RoboDK station: kr30 cnc template amana 46348 - paulina work pls TOO LOW AAA 2.rdk

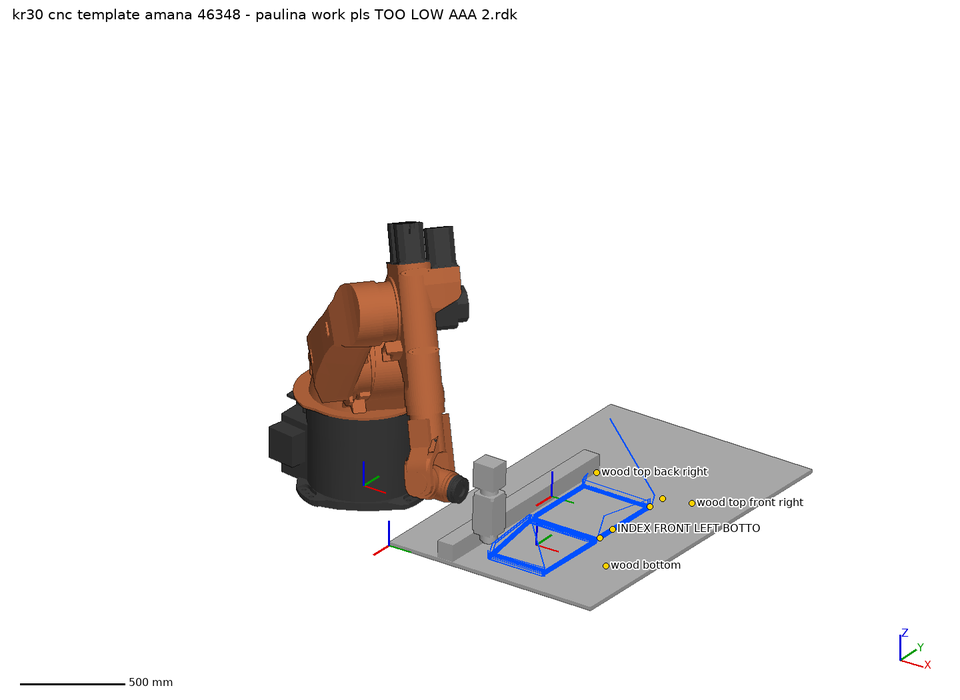
[picture v0: the station drawn from its stored meshes, robots at their saved joint values, targets as dots, program paths as lines]
Station kr30 cnc template amana 46348 - paulina work pls TOO LOW AAA 2. Poses are relative to the parent item; angles as X-Y-Z fixed-axis rotations.
  - frame KUKA KR 30 HA Base at (0, 0, 0) mm
    - robot KUKA KR 30 HA: 6 axes, payload 30 kg, reach 2033 mm, repeatability 0.05 mm, weight 665 kg
        modified DH rows (alpha deg, a mm, theta deg, d mm): 0, 0, 0, 815; -90, 350, 0, 0; 0, 850, -90, 0; -90, 145, 0, 820; 90, 0, 0, 0; -90, 0, 180, 170
        joint limits [-185, -135, -120, -350, -119, -350] to [185, 35, 158, 350, 119, 350]; home [0, -90, 90, 0, 0, 0]; saved at [41.891, -43.185, 108.764, -135.148, 71.183, 163.257]
      - tool rc90 spindle mm, TCP at (267.95, 0.68, 160.99) mm, rotated rx 0 ry 90 rz 0 deg, size 110 x 421.3 x 118 mm, geometry from rc90 spindle mm.stl
    - frame Tabletop at (921.82, -1104.91, 385) mm, rotated rx -0.93 ry -0.21 rz -89.9 deg
      - object tabletop CHECK HEIGHT at (-1839.9, 0, 0) mm, size 1839.9 x 1168.4 x 19 mm, geometry from kr30 tabletop mm.stl
      - object kr30 pipe jig base at (-1220, -610.6, 0) mm, size 1217.6 x 88.9 x 88.9 mm, geometry from kr30 pipe jig base.stl
      - frame Frame 3 at (-820, 370, 45) mm
        - frame Frame 4 at (470, 240, 0) mm, rotated rx 0 ry 0 rz 90 deg
      - target wood top back right (Cartesian target) at (-1141.49, 406.84, 52.26) mm, rotated rx 18.07 ry 89.88 rz 108.17 deg; joints [-2.086, -55.392, 143.759, 178.106, 87.553, -179.775] of KUKA KR 30 HA
      - target wood bottom (Cartesian target) at (-376.62, 995.52, 35.89) mm, rotated rx 18.07 ry 89.88 rz 108.17 deg; joints [24.587, -27.296, 76.752, 211.623, 53.064, -199.759] of KUKA KR 30 HA
      - target wood top front right (Cartesian target) at (-1142.68, 960.22, 52.55) mm, rotated rx 18.06 ry 89.88 rz 108.16 deg; joints [-1.42, -37.516, 98.016, 178.579, 59.693, -179.129] of KUKA KR 30 HA
      - target INDEX FRONT LEFT BOTTOM OF CUT (Cartesian target) at (-711.64, 800.54, 39.36) mm, rotated rx 179.19 ry 0.89 rz -118.74 deg; joints [9.3, -40.938, 107.706, -20.874, -68.324, 7.9] of KUKA KR 30 HA
      - target index front right bottom (Cartesian target) at (-1126.88, 801.86, 37.54) mm, rotated rx -179.93 ry 1.1 rz -61.86 deg; joints [5.389, -41.179, 108.718, 35.697, -71.625, -13.066] of KUKA KR 30 HA
    - target new front left bottom (Cartesian target) at (1722.92, -500.67, 408.01) mm, rotated rx 179.79 ry 0.28 rz -161.47 deg; joints [23.344, -37.525, 99.802, 45.258, -69.995, -19.505] of KUKA KR 30 HA
    - target new front right bottom (Cartesian target) at (1723.89, -86.44, 408.76) mm, rotated rx 179.79 ry 0.28 rz -161.47 deg; joints [7.822, -41.869, 110.032, 28.03, -70.804, -10.277] of KUKA KR 30 HA
  - machining project Machining Settings: C:/Users/Research Office/Desktop/paulina a5.apt | rotZ(0) | rotX(0)*rotY(0) | rotZ(0)
  - machining project Machining Settings2: C:/Users/Research Office/Desktop/paulina wooorrkkk.apt | rotZ(0) | rotX(0)*rotY(0) | rotz(0) | onStart | onPathStart | onApproach | onPoint | onRetract | onFinish | onPathFinish
  - program Machining (2349 instructions, listed below)
  - program Machining (769 instructions, listed below)
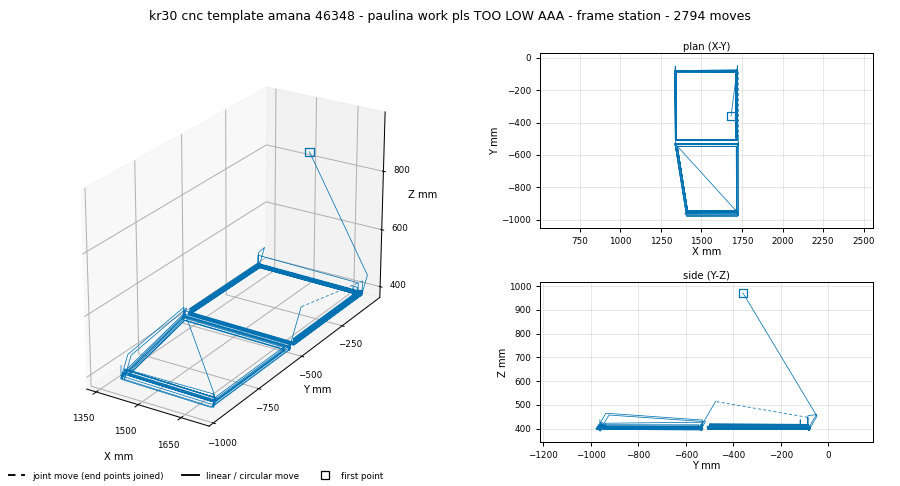
[picture p0: tool path of kr30 cnc template amana 46348 - paulina work pls TOO LOW AAA 2.rdk in frame station, 2794 of 2794 moves have a stored position in this frame; points joined in program order, loops and branches not executed]

--- program Machining (robot KUKA KR 30 HA) ---
  Smooth(15)
  Print: /'1001'
  Print: /''
  Print: /'diagonal cut'
  Set speed (100.0 mm/s)
  Set Ref.: Frame 3
  Set Tool: rc90 spindle mm
  Show rc90 spindle mm
  MoveJ 1 to (78.48, 382.25, 556.62) mm, rotated rx 174.11 ry -15.54 rz -70.77 deg; joints [17.697, -62.551, 89.928, 80.197, -35.892, -71.862]
  MoveL 2 to (-235.36, 431, 39.15) mm, rotated rx -174.06 ry -29.54 rz -11.91 deg; joints [6.63, -38.675, 85.378, -71.398, 65.68, 136.343]
  MoveL 3 to (-235.36, 431, 39.15) mm, rotated rx -174.06 ry -29.54 rz -11.91 deg; joints [6.63, -38.675, 85.378, -71.398, 65.68, 136.343]
  Set speed (100.0 mm/s)
  MoveL 4 to (-206.65, 431, -10.41) mm, rotated rx -174.06 ry -29.54 rz -11.91 deg; joints [7.609, -36.412, 85.1, -71.619, 65.676, 138.638]
  Set speed (38.1 mm/s)
  MoveL 5 to (-201.55, 431, -19.21) mm, rotated rx -174.06 ry -29.54 rz -11.91 deg; joints [7.783, -35.998, 85.023, -71.649, 65.678, 139.029]
  MoveL 6 to (-200.68, 431, -19.44) mm, rotated rx -174.06 ry -29.54 rz -11.91 deg; joints [7.812, -35.981, 85.01, -71.631, 65.695, 139.038]
  Set speed (76.2 mm/s)
  MoveL 7 to (-202.44, 431, -12.48) mm, rotated rx -174.06 ry -29.54 rz -11.91 deg; joints [7.751, -36.293, 85.037, -71.549, 65.747, 138.728]
  MoveL 8 to (-201.13, 431, -12.23) mm, rotated rx -174.06 ry -29.54 rz -11.91 deg; joints [7.795, -36.294, 85.017, -71.511, 65.781, 138.716]
  MoveL 9 to (-196.56, 431, -16.91) mm, rotated rx -174.06 ry -29.54 rz -11.91 deg; joints [7.95, -36.06, 84.947, -71.479, 65.826, 138.922]
  Set speed (38.1 mm/s)
  MoveL 10 to (-196.33, 431, -16.04) mm, rotated rx -174.06 ry -29.54 rz -11.91 deg; joints [7.958, -36.095, 84.943, -71.457, 65.843, 138.883]
  Set speed (100.0 mm/s)
  MoveL 11 to (-203.65, 431, -3.41) mm, rotated rx -174.06 ry -29.54 rz -11.91 deg; joints [7.709, -36.688, 85.05, -71.414, 65.842, 138.321]
  MoveL 12 to (-199.05, 427.82, -0.75) mm, rotated rx -174.06 ry -29.54 rz -11.91 deg; joints [7.878, -36.942, 85.328, -71.314, 65.94, 138.386]
  Set speed (38.1 mm/s)
  MoveL 13 to (-197.47, 427.82, -3.47) mm, rotated rx -174.06 ry -29.54 rz -11.91 deg; joints [7.932, -36.814, 85.306, -71.324, 65.94, 138.508]
  MoveL 14 to (-197.39, 427.82, -3.84) mm, rotated rx -174.06 ry -29.54 rz -11.91 deg; joints [7.935, -36.798, 85.305, -71.328, 65.937, 138.525]
  Set speed (76.2 mm/s)
  MoveL 15 to (-197.71, 427.82, -8.22) mm, rotated rx -174.06 ry -29.54 rz -11.91 deg; joints [7.925, -36.614, 85.314, -71.416, 65.869, 138.722]
  MoveL 16 to (-199.91, 427.82, -8.42) mm, rotated rx -174.06 ry -29.54 rz -11.91 deg; joints [7.851, -36.621, 85.348, -71.477, 65.815, 138.733]
  MoveL 17 to (-206.05, 427.82, -11.57) mm, rotated rx -174.06 ry -29.54 rz -11.91 deg; joints [7.644, -36.531, 85.443, -71.692, 65.627, 138.878]
  MoveL 18 to (-201.08, 427.82, -20.25) mm, rotated rx -174.06 ry -29.54 rz -11.91 deg; joints [7.814, -36.122, 85.367, -71.723, 65.628, 139.265]
  MoveL 19 to (-201.08, 424.65, -20.25) mm, rotated rx -174.06 ry -29.54 rz -11.91 deg; joints [7.829, -36.293, 85.717, -71.79, 65.581, 139.454]
  MoveL 20 to (-206.05, 424.65, -11.57) mm, rotated rx -174.06 ry -29.54 rz -11.91 deg; joints [7.659, -36.704, 85.792, -71.758, 65.581, 139.066]
  MoveL 21 to (-200.05, 424.65, -8.41) mm, rotated rx -174.06 ry -29.54 rz -11.91 deg; joints [7.861, -36.796, 85.7, -71.545, 65.765, 138.92]
  MoveL 22 to (-197.85, 424.65, -8.4) mm, rotated rx -174.06 ry -29.54 rz -11.91 deg; joints [7.935, -36.78, 85.666, -71.488, 65.817, 138.918]
  MoveL 23 to (-197.85, 424.65, -4.14) mm, rotated rx -174.06 ry -29.54 rz -11.91 deg; joints [7.935, -36.962, 85.662, -71.41, 65.875, 138.725]
  Set speed (38.1 mm/s)
  MoveL 24 to (-197.89, 424.65, -3.98) mm, rotated rx -174.06 ry -29.54 rz -11.91 deg; joints [7.933, -36.969, 85.663, -71.408, 65.877, 138.718]
  MoveL 25 to (-198.05, 424.33, -3.7) mm, rotated rx -174.06 ry -29.54 rz -11.91 deg; joints [7.929, -36.999, 85.7, -71.414, 65.872, 138.724]
  Set speed (76.2 mm/s)
  MoveL 26 to (-198.05, 421.79, -3.7) mm, rotated rx -174.06 ry -29.54 rz -11.91 deg; joints [7.941, -37.137, 85.979, -71.466, 65.835, 138.873]
  Set speed (38.1 mm/s)
  MoveL 27 to (-197.89, 421.47, -3.98) mm, rotated rx -174.06 ry -29.54 rz -11.91 deg; joints [7.948, -37.142, 86.011, -71.473, 65.83, 138.904]
  MoveL 28 to (-197.85, 421.47, -4.14) mm, rotated rx -174.06 ry -29.54 rz -11.91 deg; joints [7.95, -37.135, 86.011, -71.475, 65.829, 138.911]
  Set speed (76.2 mm/s)
  MoveL 29 to (-197.85, 421.47, -8.28) mm, rotated rx -174.06 ry -29.54 rz -11.91 deg; joints [7.951, -36.957, 86.014, -71.551, 65.772, 139.099]
  MoveL 30 to (-200, 421.47, -8.41) mm, rotated rx -174.06 ry -29.54 rz -11.91 deg; joints [7.878, -36.968, 86.047, -71.61, 65.72, 139.107]
  MoveL 31 to (-206.05, 421.47, -11.57) mm, rotated rx -174.06 ry -29.54 rz -11.91 deg; joints [7.673, -36.876, 86.14, -71.825, 65.535, 139.254]
  MoveL 32 to (-201.08, 421.47, -20.25) mm, rotated rx -174.06 ry -29.54 rz -11.91 deg; joints [7.844, -36.464, 86.065, -71.856, 65.535, 139.642]
  MoveL 33 to (-201.08, 418.3, -20.25) mm, rotated rx -174.06 ry -29.54 rz -11.91 deg; joints [7.859, -36.635, 86.412, -71.923, 65.489, 139.83]
  MoveL 34 to (-206.05, 418.3, -11.57) mm, rotated rx -174.06 ry -29.54 rz -11.91 deg; joints [7.688, -37.047, 86.487, -71.891, 65.489, 139.44]
  MoveL 35 to (-199.95, 418.3, -8.41) mm, rotated rx -174.06 ry -29.54 rz -11.91 deg; joints [7.895, -37.139, 86.394, -71.673, 65.675, 139.293]
  MoveL 36 to (-197.85, 418.3, -8.16) mm, rotated rx -174.06 ry -29.54 rz -11.91 deg; joints [7.966, -37.134, 86.361, -71.614, 65.728, 139.28]
  MoveL 37 to (-197.85, 418.3, -4.14) mm, rotated rx -174.06 ry -29.54 rz -11.91 deg; joints [7.965, -37.307, 86.358, -71.54, 65.783, 139.097]
  Set speed (38.1 mm/s)
  MoveL 38 to (-197.89, 418.3, -3.98) mm, rotated rx -174.06 ry -29.54 rz -11.91 deg; joints [7.963, -37.314, 86.359, -71.538, 65.784, 139.09]
  MoveL 39 to (-198.05, 417.98, -3.7) mm, rotated rx -174.06 ry -29.54 rz -11.91 deg; joints [7.96, -37.344, 86.395, -71.543, 65.779, 139.096]
  Set speed (76.2 mm/s)
  MoveL 40 to (-198.05, 415.44, -3.7) mm, rotated rx -174.06 ry -29.54 rz -11.91 deg; joints [7.972, -37.481, 86.672, -71.595, 65.743, 139.244]
  Set speed (38.1 mm/s)
  MoveL 41 to (-197.89, 415.12, -3.98) mm, rotated rx -174.06 ry -29.54 rz -11.91 deg; joints [7.979, -37.485, 86.704, -71.602, 65.738, 139.275]
  MoveL 42 to (-197.85, 415.12, -4.14) mm, rotated rx -174.06 ry -29.54 rz -11.91 deg; joints [7.98, -37.478, 86.704, -71.604, 65.737, 139.282]
  Set speed (76.2 mm/s)
  MoveL 43 to (-197.85, 415.12, -8.4) mm, rotated rx -174.06 ry -29.54 rz -11.91 deg; joints [7.981, -37.294, 86.707, -71.683, 65.679, 139.477]
  MoveL 44 to (-199.9, 415.12, -8.41) mm, rotated rx -174.06 ry -29.54 rz -11.91 deg; joints [7.911, -37.309, 86.739, -71.737, 65.631, 139.478]
  MoveL 45 to (-206.05, 415.12, -11.57) mm, rotated rx -174.06 ry -29.54 rz -11.91 deg; joints [7.703, -37.217, 86.833, -71.957, 65.444, 139.627]
  MoveL 46 to (-201.08, 415.12, -20.25) mm, rotated rx -174.06 ry -29.54 rz -11.91 deg; joints [7.874, -36.804, 86.758, -71.989, 65.444, 140.017]
  MoveL 47 to (-201.08, 411.95, -20.25) mm, rotated rx -174.06 ry -29.54 rz -11.91 deg; joints [7.889, -36.973, 87.102, -72.055, 65.399, 140.204]
  MoveL 48 to (-206.05, 411.95, -11.57) mm, rotated rx -174.06 ry -29.54 rz -11.91 deg; joints [7.718, -37.387, 87.177, -72.023, 65.399, 139.812]
  MoveL 49 to (-199.84, 411.95, -8.41) mm, rotated rx -174.06 ry -29.54 rz -11.91 deg; joints [7.928, -37.479, 87.082, -71.801, 65.587, 139.663]
  MoveL 50 to (-197.85, 411.95, -8.4) mm, rotated rx -174.06 ry -29.54 rz -11.91 deg; joints [7.996, -37.465, 87.052, -71.748, 65.634, 139.662]
  MoveL 51 to (-197.85, 411.95, -4.14) mm, rotated rx -174.06 ry -29.54 rz -11.91 deg; joints [7.996, -37.649, 87.048, -71.668, 65.692, 139.466]
  Set speed (38.1 mm/s)
  MoveL 52 to (-197.89, 411.95, -3.98) mm, rotated rx -174.06 ry -29.54 rz -11.91 deg; joints [7.994, -37.656, 87.049, -71.666, 65.693, 139.459]
  MoveL 53 to (-198.05, 411.63, -3.7) mm, rotated rx -174.06 ry -29.54 rz -11.91 deg; joints [7.99, -37.686, 87.085, -71.672, 65.689, 139.465]
  Set speed (76.2 mm/s)
  MoveL 54 to (-198.05, 409.09, -3.7) mm, rotated rx -174.06 ry -29.54 rz -11.91 deg; joints [8.002, -37.822, 87.36, -71.723, 65.653, 139.612]
  Set speed (38.1 mm/s)
  MoveL 55 to (-197.89, 408.77, -3.98) mm, rotated rx -174.06 ry -29.54 rz -11.91 deg; joints [8.009, -37.826, 87.392, -71.73, 65.648, 139.643]
  MoveL 56 to (-197.85, 408.77, -4.14) mm, rotated rx -174.06 ry -29.54 rz -11.91 deg; joints [8.011, -37.819, 87.391, -71.732, 65.647, 139.65]
  Set speed (76.2 mm/s)
  MoveL 57 to (-197.85, 408.77, -8.4) mm, rotated rx -174.06 ry -29.54 rz -11.91 deg; joints [8.012, -37.634, 87.395, -71.813, 65.589, 139.846]
  MoveL 58 to (-200.19, 408.77, -8.41) mm, rotated rx -174.06 ry -29.54 rz -11.91 deg; joints [7.932, -37.651, 87.431, -71.874, 65.534, 139.848]
  MoveL 59 to (-206.05, 408.77, -11.57) mm, rotated rx -174.06 ry -29.54 rz -11.91 deg; joints [7.733, -37.556, 87.52, -72.089, 65.355, 139.997]
  MoveL 60 to (-201.08, 408.77, -20.25) mm, rotated rx -174.06 ry -29.54 rz -11.91 deg; joints [7.904, -37.141, 87.445, -72.121, 65.355, 140.39]
  MoveL 61 to (-201.08, 405.6, -20.25) mm, rotated rx -174.06 ry -29.54 rz -11.91 deg; joints [7.919, -37.309, 87.787, -72.187, 65.311, 140.576]
  MoveL 62 to (-206.05, 405.6, -11.57) mm, rotated rx -174.06 ry -29.54 rz -11.91 deg; joints [7.747, -37.724, 87.862, -72.154, 65.31, 140.182]
  MoveL 63 to (-200.12, 405.6, -8.41) mm, rotated rx -174.06 ry -29.54 rz -11.91 deg; joints [7.949, -37.819, 87.771, -71.937, 65.491, 140.032]
  MoveL 64 to (-197.85, 405.6, -8.4) mm, rotated rx -174.06 ry -29.54 rz -11.91 deg; joints [8.027, -37.803, 87.737, -71.877, 65.544, 140.03]
  MoveL 65 to (-197.85, 405.6, -4.14) mm, rotated rx -174.06 ry -29.54 rz -11.91 deg; joints [8.026, -37.988, 87.733, -71.796, 65.602, 139.833]
  MoveL 66 to (-197.85, 405.47, -3.66) mm, rotated rx -174.06 ry -29.54 rz -11.91 deg; joints [8.027, -38.015, 87.747, -71.79, 65.607, 139.819]
  MoveL 67 to (-197.85, 405.12, -3.31) mm, rotated rx -174.06 ry -29.54 rz -11.91 deg; joints [8.029, -38.049, 87.784, -71.79, 65.607, 139.823]
  MoveL 68 to (-197.85, 404.64, -3.19) mm, rotated rx -174.06 ry -29.54 rz -11.91 deg; joints [8.031, -38.08, 87.835, -71.797, 65.602, 139.844]
  MoveL 69 to (-197.85, 403.37, -3.19) mm, rotated rx -174.06 ry -29.54 rz -11.91 deg; joints [8.037, -38.147, 87.971, -71.823, 65.585, 139.917]
  MoveL 70 to (-197.85, 402.9, -3.31) mm, rotated rx -174.06 ry -29.54 rz -11.91 deg; joints [8.039, -38.167, 88.022, -71.835, 65.576, 139.951]
  MoveL 71 to (-197.85, 402.55, -3.66) mm, rotated rx -174.06 ry -29.54 rz -11.91 deg; joints [8.041, -38.171, 88.06, -71.848, 65.567, 139.987]
  MoveL 72 to (-197.85, 402.42, -4.14) mm, rotated rx -174.06 ry -29.54 rz -11.91 deg; joints [8.042, -38.157, 88.074, -71.86, 65.558, 140.016]
  MoveL 73 to (-197.85, 402.42, -8.4) mm, rotated rx -174.06 ry -29.54 rz -11.91 deg; joints [8.043, -37.972, 88.077, -71.941, 65.5, 140.213]
  MoveL 74 to (-200.05, 402.42, -8.41) mm, rotated rx -174.06 ry -29.54 rz -11.91 deg; joints [7.967, -37.987, 88.111, -72, 65.449, 140.215]
  MoveL 75 to (-206.05, 402.42, -11.57) mm, rotated rx -174.06 ry -29.54 rz -11.91 deg; joints [7.762, -37.892, 88.202, -72.22, 65.267, 140.366]
  MoveL 76 to (-201.08, 402.42, -20.25) mm, rotated rx -174.06 ry -29.54 rz -11.91 deg; joints [7.935, -37.476, 88.128, -72.252, 65.267, 140.761]
  MoveL 77 to (-201.08, 399.25, -20.25) mm, rotated rx -174.06 ry -29.54 rz -11.91 deg; joints [7.95, -37.642, 88.467, -72.318, 65.223, 140.946]
  MoveL 78 to (-206.05, 399.25, -11.57) mm, rotated rx -174.06 ry -29.54 rz -11.91 deg; joints [7.777, -38.059, 88.541, -72.285, 65.224, 140.55]
  MoveL 79 to (-199.98, 399.25, -8.41) mm, rotated rx -174.06 ry -29.54 rz -11.91 deg; joints [7.985, -38.154, 88.449, -72.062, 65.407, 140.398]
  MoveL 80 to (-197.85, 399.25, -8.4) mm, rotated rx -174.06 ry -29.54 rz -11.91 deg; joints [8.058, -38.139, 88.416, -72.005, 65.457, 140.396]
  MoveL 81 to (-197.85, 399.25, -4.14) mm, rotated rx -174.06 ry -29.54 rz -11.91 deg; joints [8.057, -38.325, 88.413, -71.923, 65.515, 140.198]
  Set speed (38.1 mm/s)
  MoveL 82 to (-197.89, 399.25, -3.98) mm, rotated rx -174.06 ry -29.54 rz -11.91 deg; joints [8.056, -38.332, 88.414, -71.922, 65.516, 140.191]
  MoveL 83 to (-198.05, 398.93, -3.7) mm, rotated rx -174.06 ry -29.54 rz -11.91 deg; joints [8.052, -38.362, 88.45, -71.927, 65.511, 140.197]
  Set speed (76.2 mm/s)
  MoveL 84 to (-198.05, 396.39, -3.7) mm, rotated rx -174.06 ry -29.54 rz -11.91 deg; joints [8.064, -38.496, 88.72, -71.978, 65.477, 140.342]
  Set speed (38.1 mm/s)
  MoveL 85 to (-197.89, 396.07, -3.98) mm, rotated rx -174.06 ry -29.54 rz -11.91 deg; joints [8.072, -38.5, 88.752, -71.985, 65.472, 140.373]
  MoveL 86 to (-197.85, 396.07, -4.14) mm, rotated rx -174.06 ry -29.54 rz -11.91 deg; joints [8.073, -38.492, 88.751, -71.987, 65.471, 140.38]
  Set speed (76.2 mm/s)
  MoveL 87 to (-197.85, 396.07, -8.4) mm, rotated rx -174.06 ry -29.54 rz -11.91 deg; joints [8.074, -38.306, 88.755, -72.068, 65.413, 140.578]
  MoveL 88 to (-199.91, 396.07, -8.41) mm, rotated rx -174.06 ry -29.54 rz -11.91 deg; joints [8.003, -38.321, 88.786, -72.124, 65.365, 140.581]
  MoveL 89 to (-206.05, 396.07, -11.57) mm, rotated rx -174.06 ry -29.54 rz -11.91 deg; joints [7.793, -38.226, 88.879, -72.35, 65.181, 140.733]
  MoveL 90 to (-201.08, 396.07, -20.25) mm, rotated rx -174.06 ry -29.54 rz -11.91 deg; joints [7.965, -37.808, 88.805, -72.383, 65.181, 141.13]
  MoveL 91 to (-201.08, 392.9, -20.25) mm, rotated rx -174.06 ry -29.54 rz -11.91 deg; joints [7.981, -37.973, 89.142, -72.448, 65.138, 141.314]
  MoveL 92 to (-206.05, 392.9, -11.57) mm, rotated rx -174.06 ry -29.54 rz -11.91 deg; joints [7.808, -38.392, 89.216, -72.415, 65.138, 140.915]
  MoveL 93 to (-199.84, 392.9, -8.41) mm, rotated rx -174.06 ry -29.54 rz -11.91 deg; joints [8.021, -38.487, 89.122, -72.186, 65.324, 140.762]
  MoveL 94 to (-197.85, 392.9, -8.38) mm, rotated rx -174.06 ry -29.54 rz -11.91 deg; joints [8.09, -38.473, 89.091, -72.132, 65.371, 140.759]
  MoveL 95 to (-197.85, 392.9, -4.14) mm, rotated rx -174.06 ry -29.54 rz -11.91 deg; joints [8.089, -38.659, 89.088, -72.05, 65.428, 140.561]
  Set speed (38.1 mm/s)
  MoveL 96 to (-197.89, 392.9, -3.98) mm, rotated rx -174.06 ry -29.54 rz -11.91 deg; joints [8.087, -38.666, 89.089, -72.048, 65.43, 140.554]
  MoveL 97 to (-198.05, 392.58, -3.7) mm, rotated rx -174.06 ry -29.54 rz -11.91 deg; joints [8.083, -38.696, 89.124, -72.053, 65.425, 140.559]
  Set speed (76.2 mm/s)
  MoveL 98 to (-198.05, 390.04, -3.7) mm, rotated rx -174.06 ry -29.54 rz -11.91 deg; joints [8.096, -38.829, 89.393, -72.104, 65.391, 140.704]
  Set speed (38.1 mm/s)
  MoveL 99 to (-197.89, 389.72, -3.98) mm, rotated rx -174.06 ry -29.54 rz -11.91 deg; joints [8.103, -38.833, 89.424, -72.111, 65.387, 140.734]
  MoveL 100 to (-197.85, 389.72, -4.14) mm, rotated rx -174.06 ry -29.54 rz -11.91 deg; joints [8.104, -38.825, 89.424, -72.113, 65.386, 140.742]
  Set speed (76.2 mm/s)
  MoveL 101 to (-197.85, 389.72, -8.26) mm, rotated rx -174.06 ry -29.54 rz -11.91 deg; joints [8.105, -38.645, 89.427, -72.193, 65.33, 140.935]
  MoveL 102 to (-199.77, 389.72, -8.41) mm, rotated rx -174.06 ry -29.54 rz -11.91 deg; joints [8.039, -38.652, 89.456, -72.248, 65.283, 140.944]
  MoveL 103 to (-206.05, 389.72, -11.57) mm, rotated rx -174.06 ry -29.54 rz -11.91 deg; joints [7.823, -38.557, 89.551, -72.48, 65.096, 141.097]
  MoveL 104 to (-201.08, 389.72, -20.25) mm, rotated rx -174.06 ry -29.54 rz -11.91 deg; joints [7.996, -38.138, 89.477, -72.513, 65.096, 141.497]
  MoveL 105 to (-201.08, 386.55, -20.25) mm, rotated rx -174.06 ry -29.54 rz -11.91 deg; joints [8.012, -38.302, 89.811, -72.578, 65.054, 141.679]
  MoveL 106 to (-206.05, 386.55, -11.57) mm, rotated rx -174.06 ry -29.54 rz -11.91 deg; joints [7.838, -38.722, 89.885, -72.545, 65.054, 141.278]
  MoveL 107 to (-199.7, 386.55, -8.41) mm, rotated rx -174.06 ry -29.54 rz -11.91 deg; joints [8.057, -38.817, 89.79, -72.31, 65.243, 141.124]
  MoveL 108 to (-197.85, 386.55, -8.41) mm, rotated rx -174.06 ry -29.54 rz -11.91 deg; joints [8.121, -38.803, 89.762, -72.259, 65.286, 141.122]
  MoveL 109 to (-197.85, 386.55, -4.14) mm, rotated rx -174.06 ry -29.54 rz -11.91 deg; joints [8.12, -38.991, 89.758, -72.176, 65.344, 140.922]
  Set speed (38.1 mm/s)
  MoveL 110 to (-197.89, 386.55, -3.98) mm, rotated rx -174.06 ry -29.54 rz -11.91 deg; joints [8.119, -38.998, 89.759, -72.174, 65.345, 140.914]
  MoveL 111 to (-198.05, 386.23, -3.7) mm, rotated rx -174.06 ry -29.54 rz -11.91 deg; joints [8.115, -39.028, 89.794, -72.179, 65.341, 140.92]
  Set speed (76.2 mm/s)
  MoveL 112 to (-198.05, 383.69, -3.7) mm, rotated rx -174.06 ry -29.54 rz -11.91 deg; joints [8.127, -39.16, 90.061, -72.229, 65.307, 141.063]
  Set speed (38.1 mm/s)
  MoveL 113 to (-197.89, 383.37, -3.98) mm, rotated rx -174.06 ry -29.54 rz -11.91 deg; joints [8.135, -39.163, 90.092, -72.237, 65.303, 141.094]
  MoveL 114 to (-197.85, 383.37, -4.14) mm, rotated rx -174.06 ry -29.54 rz -11.91 deg; joints [8.136, -39.156, 90.092, -72.239, 65.302, 141.102]
  Set speed (76.2 mm/s)
  MoveL 115 to (-197.85, 383.37, -8.4) mm, rotated rx -174.06 ry -29.54 rz -11.91 deg; joints [8.137, -38.968, 90.095, -72.322, 65.244, 141.302]
  MoveL 116 to (-199.66, 383.37, -8.41) mm, rotated rx -174.06 ry -29.54 rz -11.91 deg; joints [8.074, -38.981, 90.122, -72.372, 65.202, 141.305]
  MoveL 117 to (-206.05, 383.37, -11.57) mm, rotated rx -174.06 ry -29.54 rz -11.91 deg; joints [7.854, -38.886, 90.218, -72.609, 65.013, 141.459]
  MoveL 118 to (-201.08, 383.37, -20.25) mm, rotated rx -174.06 ry -29.54 rz -11.91 deg; joints [8.028, -38.465, 90.145, -72.642, 65.012, 141.861]
  MoveL 119 to (-201.08, 380.2, -20.25) mm, rotated rx -174.06 ry -29.54 rz -11.91 deg; joints [8.043, -38.628, 90.477, -72.707, 64.971, 142.043]
  MoveL 120 to (-206.05, 380.2, -11.57) mm, rotated rx -174.06 ry -29.54 rz -11.91 deg; joints [7.869, -39.05, 90.55, -72.673, 64.972, 141.64]
  MoveL 121 to (-200.12, 380.2, -8.41) mm, rotated rx -174.06 ry -29.54 rz -11.91 deg; joints [8.074, -39.148, 90.461, -72.447, 65.15, 141.485]
  MoveL 122 to (-197.85, 380.2, -8.4) mm, rotated rx -174.06 ry -29.54 rz -11.91 deg; joints [8.153, -39.132, 90.427, -72.385, 65.203, 141.482]
  MoveL 123 to (-197.85, 380.2, -4.14) mm, rotated rx -174.06 ry -29.54 rz -11.91 deg; joints [8.152, -39.321, 90.424, -72.301, 65.26, 141.281]
  Set speed (38.1 mm/s)
  MoveL 124 to (-197.89, 380.2, -3.98) mm, rotated rx -174.06 ry -29.54 rz -11.91 deg; joints [8.151, -39.328, 90.424, -72.299, 65.261, 141.273]
  MoveL 125 to (-198.05, 379.88, -3.7) mm, rotated rx -174.06 ry -29.54 rz -11.91 deg; joints [8.147, -39.358, 90.459, -72.304, 65.257, 141.278]
  Set speed (76.2 mm/s)
  MoveL 126 to (-198.05, 377.34, -3.7) mm, rotated rx -174.06 ry -29.54 rz -11.91 deg; joints [8.159, -39.489, 90.724, -72.354, 65.224, 141.421]
  Set speed (38.1 mm/s)
  MoveL 127 to (-197.89, 377.02, -3.98) mm, rotated rx -174.06 ry -29.54 rz -11.91 deg; joints [8.166, -39.492, 90.755, -72.361, 65.22, 141.452]
  MoveL 128 to (-197.85, 377.02, -4.14) mm, rotated rx -174.06 ry -29.54 rz -11.91 deg; joints [8.168, -39.485, 90.755, -72.363, 65.219, 141.459]
  Set speed (76.2 mm/s)
  MoveL 129 to (-197.85, 377.02, -8.4) mm, rotated rx -174.06 ry -29.54 rz -11.91 deg; joints [8.169, -39.296, 90.758, -72.448, 65.161, 141.661]
  MoveL 130 to (-200.07, 377.02, -8.41) mm, rotated rx -174.06 ry -29.54 rz -11.91 deg; joints [8.092, -39.311, 90.791, -72.509, 65.11, 141.664]
  MoveL 131 to (-206.05, 377.02, -11.57) mm, rotated rx -174.06 ry -29.54 rz -11.91 deg; joints [7.884, -39.213, 90.881, -72.737, 64.931, 141.82]
  MoveL 132 to (-201.08, 377.02, -20.25) mm, rotated rx -174.06 ry -29.54 rz -11.91 deg; joints [8.059, -38.79, 90.808, -72.771, 64.93, 142.224]
  MoveL 133 to (-201.08, 373.85, -20.25) mm, rotated rx -174.06 ry -29.54 rz -11.91 deg; joints [8.075, -38.951, 91.137, -72.835, 64.89, 142.404]
  MoveL 134 to (-206.05, 373.85, -11.57) mm, rotated rx -174.06 ry -29.54 rz -11.91 deg; joints [7.9, -39.375, 91.211, -72.801, 64.891, 141.999]
  MoveL 135 to (-200.58, 373.85, -8.41) mm, rotated rx -174.06 ry -29.54 rz -11.91 deg; joints [8.09, -39.478, 91.129, -72.586, 65.058, 141.843]
  MoveL 136 to (-197.85, 373.85, -8.4) mm, rotated rx -174.06 ry -29.54 rz -11.91 deg; joints [8.185, -39.459, 91.088, -72.51, 65.121, 141.84]
  MoveL 137 to (-197.85, 373.85, -4.14) mm, rotated rx -174.06 ry -29.54 rz -11.91 deg; joints [8.184, -39.648, 91.084, -72.426, 65.178, 141.637]
  Set speed (38.1 mm/s)
  MoveL 138 to (-197.89, 373.85, -3.98) mm, rotated rx -174.06 ry -29.54 rz -11.91 deg; joints [8.183, -39.655, 91.085, -72.424, 65.179, 141.63]
  MoveL 139 to (-198.05, 373.53, -3.7) mm, rotated rx -174.06 ry -29.54 rz -11.91 deg; joints [8.179, -39.685, 91.12, -72.429, 65.175, 141.635]
  Set speed (76.2 mm/s)
  MoveL 140 to (-198.05, 370.99, -3.7) mm, rotated rx -174.06 ry -29.54 rz -11.91 deg; joints [8.191, -39.815, 91.383, -72.478, 65.143, 141.777]
  Set speed (38.1 mm/s)
  MoveL 141 to (-197.89, 370.67, -3.98) mm, rotated rx -174.06 ry -29.54 rz -11.91 deg; joints [8.199, -39.818, 91.414, -72.486, 65.139, 141.807]
  MoveL 142 to (-197.85, 370.67, -4.14) mm, rotated rx -174.06 ry -29.54 rz -11.91 deg; joints [8.2, -39.811, 91.413, -72.488, 65.138, 141.815]
  Set speed (76.2 mm/s)
  MoveL 143 to (-197.85, 370.67, -8.4) mm, rotated rx -174.06 ry -29.54 rz -11.91 deg; joints [8.201, -39.621, 91.416, -72.572, 65.08, 142.018]
  MoveL 144 to (-200.55, 370.67, -8.41) mm, rotated rx -174.06 ry -29.54 rz -11.91 deg; joints [8.107, -39.64, 91.457, -72.648, 65.018, 142.022]
  MoveL 145 to (-206.05, 370.67, -11.57) mm, rotated rx -174.06 ry -29.54 rz -11.91 deg; joints [7.915, -39.537, 91.539, -72.865, 64.851, 142.178]
  MoveL 146 to (-201.08, 370.67, -20.25) mm, rotated rx -174.06 ry -29.54 rz -11.91 deg; joints [8.091, -39.112, 91.466, -72.899, 64.85, 142.584]
  MoveL 147 to (-201.08, 367.5, -20.25) mm, rotated rx -174.06 ry -29.54 rz -11.91 deg; joints [8.107, -39.273, 91.794, -72.963, 64.81, 142.764]
  MoveL 148 to (-206.05, 367.5, -11.57) mm, rotated rx -174.06 ry -29.54 rz -11.91 deg; joints [7.931, -39.699, 91.867, -72.929, 64.811, 142.357]
  MoveL 149 to (-200.51, 367.5, -8.41) mm, rotated rx -174.06 ry -29.54 rz -11.91 deg; joints [8.124, -39.801, 91.784, -72.71, 64.979, 142.2]
  MoveL 150 to (-197.85, 367.5, -8.4) mm, rotated rx -174.06 ry -29.54 rz -11.91 deg; joints [8.217, -39.783, 91.744, -72.635, 65.04, 142.196]
  MoveL 151 to (-197.85, 367.5, -4.14) mm, rotated rx -174.06 ry -29.54 rz -11.91 deg; joints [8.216, -39.973, 91.741, -72.549, 65.098, 141.992]
  MoveL 152 to (-197.85, 367.37, -3.66) mm, rotated rx -174.06 ry -29.54 rz -11.91 deg; joints [8.217, -40.001, 91.753, -72.542, 65.103, 141.976]
  MoveL 153 to (-197.85, 367.02, -3.31) mm, rotated rx -174.06 ry -29.54 rz -11.91 deg; joints [8.219, -40.034, 91.789, -72.542, 65.103, 141.979]
  MoveL 154 to (-197.85, 366.55, -3.19) mm, rotated rx -174.06 ry -29.54 rz -11.91 deg; joints [8.221, -40.064, 91.838, -72.549, 65.099, 142]
  MoveL 155 to (-197.85, 365.28, -3.19) mm, rotated rx -174.06 ry -29.54 rz -11.91 deg; joints [8.227, -40.129, 91.968, -72.574, 65.083, 142.07]
  MoveL 156 to (-197.85, 364.8, -3.31) mm, rotated rx -174.06 ry -29.54 rz -11.91 deg; joints [8.23, -40.147, 92.018, -72.585, 65.075, 142.103]
  MoveL 157 to (-197.85, 364.45, -3.66) mm, rotated rx -174.06 ry -29.54 rz -11.91 deg; joints [8.232, -40.15, 92.054, -72.599, 65.066, 142.139]
  MoveL 158 to (-197.85, 364.33, -4.14) mm, rotated rx -174.06 ry -29.54 rz -11.91 deg; joints [8.233, -40.135, 92.067, -72.611, 65.058, 142.169]
  MoveL 159 to (-197.85, 364.33, -8.4) mm, rotated rx -174.06 ry -29.54 rz -11.91 deg; joints [8.233, -39.944, 92.07, -72.697, 65.001, 142.373]
  MoveL 160 to (-200.48, 364.33, -8.41) mm, rotated rx -174.06 ry -29.54 rz -11.91 deg; joints [8.141, -39.962, 92.11, -72.771, 64.94, 142.377]
  MoveL 161 to (-206.05, 364.33, -11.57) mm, rotated rx -174.06 ry -29.54 rz -11.91 deg; joints [7.947, -39.859, 92.193, -72.992, 64.772, 142.535]
  MoveL 162 to (-201.08, 364.33, -20.25) mm, rotated rx -174.06 ry -29.54 rz -11.91 deg; joints [8.123, -39.433, 92.12, -73.026, 64.771, 142.943]
  MoveL 163 to (-201.08, 361.15, -20.25) mm, rotated rx -174.06 ry -29.54 rz -11.91 deg; joints [8.139, -39.592, 92.445, -73.09, 64.732, 143.122]
  MoveL 164 to (-206.05, 361.15, -11.57) mm, rotated rx -174.06 ry -29.54 rz -11.91 deg; joints [7.962, -40.02, 92.518, -73.055, 64.733, 142.712]
  MoveL 165 to (-200.44, 361.15, -8.41) mm, rotated rx -174.06 ry -29.54 rz -11.91 deg; joints [8.159, -40.123, 92.435, -72.832, 64.902, 142.554]
  MoveL 166 to (-197.85, 361.15, -8.4) mm, rotated rx -174.06 ry -29.54 rz -11.91 deg; joints [8.25, -40.105, 92.396, -72.759, 64.961, 142.55]
  MoveL 167 to (-197.85, 361.15, -4.14) mm, rotated rx -174.06 ry -29.54 rz -11.91 deg; joints [8.249, -40.296, 92.393, -72.673, 65.018, 142.345]
  Set speed (38.1 mm/s)
  MoveL 168 to (-197.89, 361.15, -3.98) mm, rotated rx -174.06 ry -29.54 rz -11.91 deg; joints [8.247, -40.303, 92.393, -72.671, 65.02, 142.337]
  MoveL 169 to (-198.05, 360.83, -3.7) mm, rotated rx -174.06 ry -29.54 rz -11.91 deg; joints [8.243, -40.333, 92.428, -72.676, 65.016, 142.342]
  Set speed (76.2 mm/s)
  MoveL 170 to (-198.05, 358.29, -3.7) mm, rotated rx -174.06 ry -29.54 rz -11.91 deg; joints [8.256, -40.462, 92.687, -72.725, 64.984, 142.483]
  Set speed (38.1 mm/s)
  MoveL 171 to (-197.89, 357.98, -3.98) mm, rotated rx -174.06 ry -29.54 rz -11.91 deg; joints [8.264, -40.464, 92.718, -72.732, 64.981, 142.513]
  MoveL 172 to (-197.85, 357.98, -4.14) mm, rotated rx -174.06 ry -29.54 rz -11.91 deg; joints [8.265, -40.457, 92.717, -72.734, 64.979, 142.521]
  Set speed (76.2 mm/s)
  MoveL 173 to (-197.85, 357.98, -8.25) mm, rotated rx -174.06 ry -29.54 rz -11.91 deg; joints [8.266, -40.272, 92.72, -72.817, 64.924, 142.719]
  MoveL 174 to (-200.41, 357.98, -8.41) mm, rotated rx -174.06 ry -29.54 rz -11.91 deg; joints [8.176, -40.283, 92.759, -72.893, 64.864, 142.73]
  MoveL 175 to (-206.05, 357.98, -11.57) mm, rotated rx -174.06 ry -29.54 rz -11.91 deg; joints [7.978, -40.179, 92.843, -73.118, 64.694, 142.889]
  MoveL 176 to (-201.08, 357.98, -20.25) mm, rotated rx -174.06 ry -29.54 rz -11.91 deg; joints [8.155, -39.751, 92.77, -73.153, 64.693, 143.3]
  MoveL 177 to (-201.08, 354.8, -20.25) mm, rotated rx -174.06 ry -29.54 rz -11.91 deg; joints [8.171, -39.909, 93.093, -73.216, 64.655, 143.478]
  MoveL 178 to (-206.05, 354.8, -11.57) mm, rotated rx -174.06 ry -29.54 rz -11.91 deg; joints [7.994, -40.339, 93.166, -73.181, 64.656, 143.066]
  MoveL 179 to (-200.37, 354.8, -8.41) mm, rotated rx -174.06 ry -29.54 rz -11.91 deg; joints [8.193, -40.442, 93.081, -72.954, 64.826, 142.906]
  MoveL 180 to (-197.85, 354.8, -8.13) mm, rotated rx -174.06 ry -29.54 rz -11.91 deg; joints [8.282, -40.437, 93.043, -72.877, 64.887, 142.889]
  MoveL 181 to (-197.85, 354.8, -4.14) mm, rotated rx -174.06 ry -29.54 rz -11.91 deg; joints [8.282, -40.617, 93.04, -72.795, 64.941, 142.696]
  MoveL 182 to (-197.85, 354.67, -3.66) mm, rotated rx -174.06 ry -29.54 rz -11.91 deg; joints [8.282, -40.645, 93.053, -72.788, 64.945, 142.68]
  MoveL 183 to (-197.85, 354.32, -3.31) mm, rotated rx -174.06 ry -29.54 rz -11.91 deg; joints [8.284, -40.678, 93.088, -72.788, 64.946, 142.682]
  MoveL 184 to (-197.85, 353.85, -3.19) mm, rotated rx -174.06 ry -29.54 rz -11.91 deg; joints [8.286, -40.708, 93.136, -72.794, 64.942, 142.702]
  MoveL 185 to (-197.85, 352.58, -3.19) mm, rotated rx -174.06 ry -29.54 rz -11.91 deg; joints [8.293, -40.771, 93.265, -72.819, 64.926, 142.772]
  MoveL 186 to (-197.85, 352.1, -3.31) mm, rotated rx -174.06 ry -29.54 rz -11.91 deg; joints [8.295, -40.79, 93.314, -72.83, 64.919, 142.805]
  MoveL 187 to (-197.85, 351.75, -3.66) mm, rotated rx -174.06 ry -29.54 rz -11.91 deg; joints [8.297, -40.791, 93.349, -72.844, 64.91, 142.841]
  MoveL 188 to (-197.85, 351.63, -4.14) mm, rotated rx -174.06 ry -29.54 rz -11.91 deg; joints [8.298, -40.776, 93.363, -72.856, 64.902, 142.871]
  MoveL 189 to (-197.85, 351.63, -8.4) mm, rotated rx -174.06 ry -29.54 rz -11.91 deg; joints [8.299, -40.584, 93.366, -72.944, 64.845, 143.078]
  MoveL 190 to (-200.34, 351.63, -8.41) mm, rotated rx -174.06 ry -29.54 rz -11.91 deg; joints [8.211, -40.601, 93.403, -73.015, 64.788, 143.082]
  MoveL 191 to (-206.05, 351.63, -11.57) mm, rotated rx -174.06 ry -29.54 rz -11.91 deg; joints [8.01, -40.497, 93.488, -73.244, 64.618, 143.242]
  MoveL 192 to (-201.08, 351.63, -20.25) mm, rotated rx -174.06 ry -29.54 rz -11.91 deg; joints [8.187, -40.067, 93.415, -73.279, 64.616, 143.656]
  MoveL 193 to (-201.08, 348.45, -20.25) mm, rotated rx -174.06 ry -29.54 rz -11.91 deg; joints [8.204, -40.224, 93.736, -73.342, 64.579, 143.833]
  MoveL 194 to (-206.05, 348.45, -11.57) mm, rotated rx -174.06 ry -29.54 rz -11.91 deg; joints [8.026, -40.655, 93.809, -73.307, 64.58, 143.418]
  MoveL 195 to (-199.95, 348.45, -8.41) mm, rotated rx -174.06 ry -29.54 rz -11.91 deg; joints [8.241, -40.757, 93.718, -73.066, 64.759, 143.256]
  MoveL 196 to (-197.85, 348.45, -8.4) mm, rotated rx -174.06 ry -29.54 rz -11.91 deg; joints [8.316, -40.742, 93.687, -73.005, 64.807, 143.253]
  MoveL 197 to (-197.85, 348.45, -4.14) mm, rotated rx -174.06 ry -29.54 rz -11.91 deg; joints [8.315, -40.935, 93.684, -72.917, 64.864, 143.045]
  MoveL 198 to (-197.85, 348.32, -3.66) mm, rotated rx -174.06 ry -29.54 rz -11.91 deg; joints [8.315, -40.963, 93.696, -72.91, 64.869, 143.029]
  MoveL 199 to (-197.85, 347.98, -3.31) mm, rotated rx -174.06 ry -29.54 rz -11.91 deg; joints [8.317, -40.997, 93.731, -72.909, 64.869, 143.031]
  MoveL 200 to (-197.85, 347.5, -3.19) mm, rotated rx -174.06 ry -29.54 rz -11.91 deg; joints [8.319, -41.026, 93.779, -72.916, 64.865, 143.051]
  MoveL 201 to (-197.85, 346.23, -3.19) mm, rotated rx -174.06 ry -29.54 rz -11.91 deg; joints [8.326, -41.09, 93.907, -72.94, 64.85, 143.121]
  MoveL 202 to (-197.85, 345.75, -3.31) mm, rotated rx -174.06 ry -29.54 rz -11.91 deg; joints [8.329, -41.108, 93.955, -72.952, 64.843, 143.153]
  MoveL 203 to (-197.85, 345.4, -3.66) mm, rotated rx -174.06 ry -29.54 rz -11.91 deg; joints [8.33, -41.109, 93.991, -72.966, 64.834, 143.189]
  MoveL 204 to (-197.85, 345.28, -4.14) mm, rotated rx -174.06 ry -29.54 rz -11.91 deg; joints [8.331, -41.094, 94.004, -72.978, 64.826, 143.219]
  MoveL 205 to (-197.85, 345.28, -8.4) mm, rotated rx -174.06 ry -29.54 rz -11.91 deg; joints [8.332, -40.9, 94.007, -73.066, 64.769, 143.428]
  MoveL 206 to (-199.91, 345.28, -8.41) mm, rotated rx -174.06 ry -29.54 rz -11.91 deg; joints [8.259, -40.915, 94.038, -73.126, 64.722, 143.431]
  MoveL 207 to (-206.05, 345.28, -11.57) mm, rotated rx -174.06 ry -29.54 rz -11.91 deg; joints [8.042, -40.813, 94.129, -73.369, 64.543, 143.594]
  MoveL 208 to (-201.08, 345.28, -20.25) mm, rotated rx -174.06 ry -29.54 rz -11.91 deg; joints [8.22, -40.381, 94.056, -73.405, 64.541, 144.009]
  MoveL 209 to (-201.08, 342.1, -20.25) mm, rotated rx -174.06 ry -29.54 rz -11.91 deg; joints [8.237, -40.537, 94.376, -73.467, 64.504, 144.185]
  MoveL 210 to (-206.05, 342.1, -11.57) mm, rotated rx -174.06 ry -29.54 rz -11.91 deg; joints [8.058, -40.97, 94.448, -73.431, 64.506, 143.769]
  MoveL 211 to (-199.87, 342.1, -8.41) mm, rotated rx -174.06 ry -29.54 rz -11.91 deg; joints [8.277, -41.072, 94.357, -73.186, 64.686, 143.605]
  MoveL 212 to (-197.85, 342.1, -8.4) mm, rotated rx -174.06 ry -29.54 rz -11.91 deg; joints [8.349, -41.058, 94.327, -73.127, 64.732, 143.602]
  MoveL 213 to (-197.85, 342.1, -4.14) mm, rotated rx -174.06 ry -29.54 rz -11.91 deg; joints [8.348, -41.252, 94.323, -73.038, 64.789, 143.393]
  Set speed (38.1 mm/s)
  MoveL 214 to (-197.89, 342.1, -3.98) mm, rotated rx -174.06 ry -29.54 rz -11.91 deg; joints [8.346, -41.26, 94.324, -73.036, 64.79, 143.385]
  MoveL 215 to (-198.05, 341.78, -3.7) mm, rotated rx -174.06 ry -29.54 rz -11.91 deg; joints [8.342, -41.289, 94.358, -73.041, 64.786, 143.389]
  Set speed (76.2 mm/s)
  MoveL 216 to (-198.05, 339.25, -3.7) mm, rotated rx -174.06 ry -29.54 rz -11.91 deg; joints [8.356, -41.415, 94.612, -73.09, 64.757, 143.528]
  Set speed (38.1 mm/s)
  MoveL 217 to (-197.89, 338.93, -3.98) mm, rotated rx -174.06 ry -29.54 rz -11.91 deg; joints [8.363, -41.417, 94.642, -73.097, 64.753, 143.558]
  MoveL 218 to (-197.85, 338.93, -4.14) mm, rotated rx -174.06 ry -29.54 rz -11.91 deg; joints [8.365, -41.41, 94.642, -73.099, 64.752, 143.566]
  Set speed (76.2 mm/s)
  MoveL 219 to (-197.85, 338.93, -8.4) mm, rotated rx -174.06 ry -29.54 rz -11.91 deg; joints [8.366, -41.215, 94.645, -73.188, 64.695, 143.776]
  MoveL 220 to (-200.2, 338.93, -8.41) mm, rotated rx -174.06 ry -29.54 rz -11.91 deg; joints [8.282, -41.231, 94.68, -73.257, 64.642, 143.779]
  MoveL 221 to (-206.05, 338.93, -11.57) mm, rotated rx -174.06 ry -29.54 rz -11.91 deg; joints [8.074, -41.127, 94.766, -73.494, 64.469, 143.943]
  MoveL 222 to (-201.08, 338.93, -20.25) mm, rotated rx -174.06 ry -29.54 rz -11.91 deg; joints [8.253, -40.693, 94.694, -73.529, 64.467, 144.361]
  MoveL 223 to (-201.08, 335.75, -20.25) mm, rotated rx -174.06 ry -29.54 rz -11.91 deg; joints [8.27, -40.848, 95.011, -73.592, 64.431, 144.536]
  MoveL 224 to (-206.05, 335.75, -11.57) mm, rotated rx -174.06 ry -29.54 rz -11.91 deg; joints [8.091, -41.283, 95.083, -73.556, 64.432, 144.117]
  MoveL 225 to (-200.15, 335.75, -8.41) mm, rotated rx -174.06 ry -29.54 rz -11.91 deg; joints [8.3, -41.388, 94.996, -73.316, 64.606, 143.953]
  MoveL 226 to (-197.85, 335.75, -8.4) mm, rotated rx -174.06 ry -29.54 rz -11.91 deg; joints [8.382, -41.372, 94.962, -73.248, 64.658, 143.949]
  MoveL 227 to (-197.85, 335.75, -4.14) mm, rotated rx -174.06 ry -29.54 rz -11.91 deg; joints [8.381, -41.567, 94.959, -73.159, 64.715, 143.739]
  Set speed (38.1 mm/s)
  MoveL 228 to (-197.89, 335.75, -3.98) mm, rotated rx -174.06 ry -29.54 rz -11.91 deg; joints [8.38, -41.574, 94.959, -73.157, 64.716, 143.731]
  MoveL 229 to (-198.05, 335.44, -3.7) mm, rotated rx -174.06 ry -29.54 rz -11.91 deg; joints [8.376, -41.604, 94.993, -73.162, 64.712, 143.735]
  Set speed (76.2 mm/s)
  MoveL 230 to (-198.05, 332.9, -3.7) mm, rotated rx -174.06 ry -29.54 rz -11.91 deg; joints [8.389, -41.729, 95.246, -73.21, 64.683, 143.873]
  Set speed (38.1 mm/s)
  MoveL 231 to (-197.89, 332.58, -3.98) mm, rotated rx -174.06 ry -29.54 rz -11.91 deg; joints [8.397, -41.731, 95.276, -73.217, 64.679, 143.903]
  MoveL 232 to (-197.85, 332.58, -4.14) mm, rotated rx -174.06 ry -29.54 rz -11.91 deg; joints [8.398, -41.723, 95.275, -73.219, 64.678, 143.911]
  Set speed (76.2 mm/s)
  MoveL 233 to (-197.85, 332.58, -8.4) mm, rotated rx -174.06 ry -29.54 rz -11.91 deg; joints [8.399, -41.528, 95.278, -73.309, 64.621, 144.122]
  MoveL 234 to (-200.15, 332.58, -8.41) mm, rotated rx -174.06 ry -29.54 rz -11.91 deg; joints [8.317, -41.544, 95.312, -73.377, 64.57, 144.126]
  MoveL 235 to (-206.05, 332.58, -11.57) mm, rotated rx -174.06 ry -29.54 rz -11.91 deg; joints [8.107, -41.439, 95.399, -73.617, 64.396, 144.291]
  MoveL 236 to (-201.08, 332.58, -20.25) mm, rotated rx -174.06 ry -29.54 rz -11.91 deg; joints [8.286, -41.003, 95.327, -73.654, 64.395, 144.711]
  MoveL 237 to (-201.08, 329.4, -20.25) mm, rotated rx -174.06 ry -29.54 rz -11.91 deg; joints [8.303, -41.157, 95.642, -73.715, 64.359, 144.885]
  MoveL 238 to (-206.05, 329.4, -11.57) mm, rotated rx -174.06 ry -29.54 rz -11.91 deg; joints [8.123, -41.594, 95.715, -73.679, 64.36, 144.464]
  MoveL 239 to (-200.15, 329.4, -8.41) mm, rotated rx -174.06 ry -29.54 rz -11.91 deg; joints [8.334, -41.699, 95.628, -73.437, 64.533, 144.298]
  MoveL 240 to (-197.85, 329.4, -8.4) mm, rotated rx -174.06 ry -29.54 rz -11.91 deg; joints [8.416, -41.683, 95.594, -73.369, 64.585, 144.295]
  MoveL 241 to (-197.85, 329.4, -4.14) mm, rotated rx -174.06 ry -29.54 rz -11.91 deg; joints [8.415, -41.88, 95.59, -73.279, 64.642, 144.083]
  Set speed (38.1 mm/s)
  MoveL 242 to (-197.89, 329.4, -3.98) mm, rotated rx -174.06 ry -29.54 rz -11.91 deg; joints [8.414, -41.887, 95.591, -73.277, 64.643, 144.075]
  MoveL 243 to (-198.05, 329.09, -3.7) mm, rotated rx -174.06 ry -29.54 rz -11.91 deg; joints [8.41, -41.917, 95.624, -73.282, 64.64, 144.079]
  Set speed (76.2 mm/s)
  MoveL 244 to (-198.05, 326.55, -3.7) mm, rotated rx -174.06 ry -29.54 rz -11.91 deg; joints [8.423, -42.041, 95.876, -73.33, 64.611, 144.216]
  Set speed (38.1 mm/s)
  MoveL 245 to (-197.89, 326.23, -3.98) mm, rotated rx -174.06 ry -29.54 rz -11.91 deg; joints [8.431, -42.043, 95.905, -73.337, 64.607, 144.246]
  MoveL 246 to (-197.85, 326.23, -4.14) mm, rotated rx -174.06 ry -29.54 rz -11.91 deg; joints [8.432, -42.035, 95.905, -73.339, 64.606, 144.254]
  Set speed (76.2 mm/s)
  MoveL 247 to (-197.85, 326.23, -8.4) mm, rotated rx -174.06 ry -29.54 rz -11.91 deg; joints [8.433, -41.839, 95.908, -73.429, 64.549, 144.467]
  MoveL 248 to (-200.15, 326.23, -8.41) mm, rotated rx -174.06 ry -29.54 rz -11.91 deg; joints [8.351, -41.854, 95.942, -73.498, 64.498, 144.471]
  MoveL 249 to (-206.05, 326.23, -11.57) mm, rotated rx -174.06 ry -29.54 rz -11.91 deg; joints [8.14, -41.749, 96.029, -73.741, 64.325, 144.637]
  MoveL 250 to (-201.08, 326.23, -20.25) mm, rotated rx -174.06 ry -29.54 rz -11.91 deg; joints [8.32, -41.31, 95.957, -73.777, 64.323, 145.059]
  MoveL 251 to (-201.08, 323.05, -20.25) mm, rotated rx -174.06 ry -29.54 rz -11.91 deg; joints [8.337, -41.464, 96.27, -73.839, 64.288, 145.233]
  MoveL 252 to (-206.05, 323.05, -11.57) mm, rotated rx -174.06 ry -29.54 rz -11.91 deg; joints [8.156, -41.903, 96.342, -73.802, 64.29, 144.809]
  MoveL 253 to (-200.15, 323.05, -8.41) mm, rotated rx -174.06 ry -29.54 rz -11.91 deg; joints [8.367, -42.009, 96.255, -73.558, 64.462, 144.642]
  MoveL 254 to (-197.85, 323.05, -8.4) mm, rotated rx -174.06 ry -29.54 rz -11.91 deg; joints [8.45, -41.993, 96.221, -73.489, 64.514, 144.638]
  MoveL 255 to (-197.85, 323.05, -4.14) mm, rotated rx -174.06 ry -29.54 rz -11.91 deg; joints [8.449, -42.19, 96.218, -73.398, 64.57, 144.425]
  Set speed (38.1 mm/s)
  MoveL 256 to (-197.89, 323.05, -3.98) mm, rotated rx -174.06 ry -29.54 rz -11.91 deg; joints [8.448, -42.198, 96.219, -73.396, 64.571, 144.417]
  MoveL 257 to (-198.05, 322.74, -3.7) mm, rotated rx -174.06 ry -29.54 rz -11.91 deg; joints [8.444, -42.227, 96.252, -73.401, 64.568, 144.421]
  Set speed (76.2 mm/s)
  MoveL 258 to (-198.05, 320.2, -3.7) mm, rotated rx -174.06 ry -29.54 rz -11.91 deg; joints [8.457, -42.351, 96.502, -73.449, 64.54, 144.557]
  Set speed (38.1 mm/s)
  MoveL 259 to (-197.89, 319.88, -3.98) mm, rotated rx -174.06 ry -29.54 rz -11.91 deg; joints [8.465, -42.353, 96.531, -73.456, 64.536, 144.588]
  MoveL 260 to (-197.85, 319.88, -4.14) mm, rotated rx -174.06 ry -29.54 rz -11.91 deg; joints [8.467, -42.345, 96.531, -73.458, 64.535, 144.596]
  Set speed (76.2 mm/s)
  MoveL 261 to (-197.85, 319.88, -8.4) mm, rotated rx -174.06 ry -29.54 rz -11.91 deg; joints [8.467, -42.147, 96.534, -73.549, 64.478, 144.81]
  MoveL 262 to (-200.15, 319.88, -8.41) mm, rotated rx -174.06 ry -29.54 rz -11.91 deg; joints [8.384, -42.163, 96.568, -73.618, 64.427, 144.814]
  MoveL 263 to (-206.05, 319.88, -11.57) mm, rotated rx -174.06 ry -29.54 rz -11.91 deg; joints [8.173, -42.057, 96.655, -73.863, 64.255, 144.981]
  MoveL 264 to (-201.08, 319.88, -20.25) mm, rotated rx -174.06 ry -29.54 rz -11.91 deg; joints [8.354, -41.617, 96.583, -73.9, 64.253, 145.406]
  MoveL 265 to (-201.08, 316.7, -20.25) mm, rotated rx -174.06 ry -29.54 rz -11.91 deg; joints [8.371, -41.769, 96.894, -73.961, 64.218, 145.579]
  MoveL 266 to (-206.05, 316.7, -11.57) mm, rotated rx -174.06 ry -29.54 rz -11.91 deg; joints [8.19, -42.21, 96.966, -73.924, 64.22, 145.153]
  MoveL 267 to (-200.15, 316.7, -8.41) mm, rotated rx -174.06 ry -29.54 rz -11.91 deg; joints [8.402, -42.317, 96.879, -73.678, 64.392, 144.985]
  MoveL 268 to (-197.85, 316.7, -8.4) mm, rotated rx -174.06 ry -29.54 rz -11.91 deg; joints [8.485, -42.301, 96.845, -73.609, 64.443, 144.981]
  MoveL 269 to (-197.85, 316.7, -4.14) mm, rotated rx -174.06 ry -29.54 rz -11.91 deg; joints [8.484, -42.5, 96.842, -73.517, 64.5, 144.766]
  Set speed (38.1 mm/s)
  MoveL 270 to (-197.89, 316.7, -3.98) mm, rotated rx -174.06 ry -29.54 rz -11.91 deg; joints [8.482, -42.507, 96.843, -73.515, 64.501, 144.758]
  MoveL 271 to (-198.05, 316.39, -3.7) mm, rotated rx -174.06 ry -29.54 rz -11.91 deg; joints [8.478, -42.536, 96.876, -73.52, 64.498, 144.762]
  Set speed (76.2 mm/s)
  MoveL 272 to (-198.05, 313.85, -3.7) mm, rotated rx -174.06 ry -29.54 rz -11.91 deg; joints [8.492, -42.66, 97.124, -73.567, 64.47, 144.897]
  Set speed (38.1 mm/s)
  MoveL 273 to (-197.89, 313.53, -3.98) mm, rotated rx -174.06 ry -29.54 rz -11.91 deg; joints [8.499, -42.661, 97.153, -73.574, 64.466, 144.928]
  MoveL 274 to (-197.85, 313.53, -4.14) mm, rotated rx -174.06 ry -29.54 rz -11.91 deg; joints [8.501, -42.653, 97.153, -73.576, 64.465, 144.936]
  Set speed (76.2 mm/s)
  MoveL 275 to (-197.85, 313.53, -8.4) mm, rotated rx -174.06 ry -29.54 rz -11.91 deg; joints [8.502, -42.455, 97.156, -73.668, 64.409, 145.151]
  MoveL 276 to (-200.15, 313.53, -8.41) mm, rotated rx -174.06 ry -29.54 rz -11.91 deg; joints [8.419, -42.47, 97.19, -73.738, 64.357, 145.155]
  MoveL 277 to (-206.05, 313.53, -11.57) mm, rotated rx -174.06 ry -29.54 rz -11.91 deg; joints [8.206, -42.363, 97.277, -73.985, 64.186, 145.324]
  MoveL 278 to (-201.08, 313.53, -20.25) mm, rotated rx -174.06 ry -29.54 rz -11.91 deg; joints [8.388, -41.921, 97.205, -74.022, 64.184, 145.752]
  MoveL 279 to (-201.08, 310.35, -20.25) mm, rotated rx -174.06 ry -29.54 rz -11.91 deg; joints [8.405, -42.072, 97.515, -74.083, 64.15, 145.924]
  MoveL 280 to (-206.05, 310.35, -11.57) mm, rotated rx -174.06 ry -29.54 rz -11.91 deg; joints [8.223, -42.515, 97.586, -74.046, 64.152, 145.495]
  MoveL 281 to (-200.15, 310.35, -8.41) mm, rotated rx -174.06 ry -29.54 rz -11.91 deg; joints [8.436, -42.623, 97.5, -73.798, 64.323, 145.326]
  MoveL 282 to (-197.85, 310.35, -8.4) mm, rotated rx -174.06 ry -29.54 rz -11.91 deg; joints [8.519, -42.607, 97.466, -73.728, 64.374, 145.321]
  MoveL 283 to (-197.85, 310.35, -4.14) mm, rotated rx -174.06 ry -29.54 rz -11.91 deg; joints [8.518, -42.807, 97.463, -73.635, 64.431, 145.105]
  Set speed (38.1 mm/s)
  MoveL 284 to (-197.89, 310.35, -3.98) mm, rotated rx -174.06 ry -29.54 rz -11.91 deg; joints [8.517, -42.814, 97.463, -73.633, 64.432, 145.097]
  MoveL 285 to (-198.05, 310.04, -3.7) mm, rotated rx -174.06 ry -29.54 rz -11.91 deg; joints [8.513, -42.844, 97.496, -73.638, 64.428, 145.101]
  Set speed (76.2 mm/s)
  MoveL 286 to (-198.05, 307.5, -3.7) mm, rotated rx -174.06 ry -29.54 rz -11.91 deg; joints [8.527, -42.966, 97.743, -73.685, 64.401, 145.236]
  Set speed (38.1 mm/s)
  MoveL 287 to (-197.89, 307.18, -3.98) mm, rotated rx -174.06 ry -29.54 rz -11.91 deg; joints [8.534, -42.967, 97.772, -73.692, 64.398, 145.266]
  MoveL 288 to (-197.85, 307.18, -4.14) mm, rotated rx -174.06 ry -29.54 rz -11.91 deg; joints [8.536, -42.96, 97.772, -73.694, 64.396, 145.274]
  Set speed (76.2 mm/s)
  MoveL 289 to (-197.85, 307.18, -8.4) mm, rotated rx -174.06 ry -29.54 rz -11.91 deg; joints [8.537, -42.76, 97.775, -73.787, 64.34, 145.491]
  MoveL 290 to (-200.15, 307.18, -8.41) mm, rotated rx -174.06 ry -29.54 rz -11.91 deg; joints [8.453, -42.776, 97.809, -73.857, 64.289, 145.495]
  MoveL 291 to (-206.05, 307.18, -11.57) mm, rotated rx -174.06 ry -29.54 rz -11.91 deg; joints [8.24, -42.667, 97.895, -74.106, 64.118, 145.666]
  MoveL 292 to (-201.08, 307.18, -20.25) mm, rotated rx -174.06 ry -29.54 rz -11.91 deg; joints [8.422, -42.223, 97.823, -74.144, 64.116, 146.096]
  MoveL 293 to (-201.08, 304.01, -20.25) mm, rotated rx -174.06 ry -29.54 rz -11.91 deg; joints [8.439, -42.374, 98.131, -74.204, 64.082, 146.267]
  MoveL 294 to (-206.05, 304.01, -11.57) mm, rotated rx -174.06 ry -29.54 rz -11.91 deg; joints [8.257, -42.819, 98.203, -74.167, 64.085, 145.836]
  MoveL 295 to (-200.15, 304.01, -8.41) mm, rotated rx -174.06 ry -29.54 rz -11.91 deg; joints [8.47, -42.928, 98.117, -73.917, 64.255, 145.665]
  MoveL 296 to (-197.85, 304.01, -8.4) mm, rotated rx -174.06 ry -29.54 rz -11.91 deg; joints [8.554, -42.912, 98.083, -73.846, 64.306, 145.66]
  MoveL 297 to (-197.85, 304.01, -4.14) mm, rotated rx -174.06 ry -29.54 rz -11.91 deg; joints [8.553, -43.112, 98.08, -73.753, 64.362, 145.443]
  Set speed (38.1 mm/s)
  MoveL 298 to (-197.89, 304.01, -3.98) mm, rotated rx -174.06 ry -29.54 rz -11.91 deg; joints [8.552, -43.12, 98.08, -73.75, 64.364, 145.435]
  MoveL 299 to (-198.05, 303.69, -3.7) mm, rotated rx -174.06 ry -29.54 rz -11.91 deg; joints [8.548, -43.149, 98.113, -73.755, 64.36, 145.438]
  Set speed (76.2 mm/s)
  MoveL 300 to (-198.05, 301.15, -3.7) mm, rotated rx -174.06 ry -29.54 rz -11.91 deg; joints [8.562, -43.271, 98.359, -73.802, 64.333, 145.573]
  Set speed (38.1 mm/s)
  MoveL 301 to (-197.89, 300.83, -3.98) mm, rotated rx -174.06 ry -29.54 rz -11.91 deg; joints [8.569, -43.272, 98.387, -73.809, 64.33, 145.603]
  MoveL 302 to (-197.85, 300.83, -4.14) mm, rotated rx -174.06 ry -29.54 rz -11.91 deg; joints [8.571, -43.264, 98.387, -73.811, 64.329, 145.611]
  Set speed (76.2 mm/s)
  MoveL 303 to (-197.85, 300.83, -8.4) mm, rotated rx -174.06 ry -29.54 rz -11.91 deg; joints [8.572, -43.063, 98.39, -73.905, 64.273, 145.829]
  MoveL 304 to (-200.15, 300.83, -8.41) mm, rotated rx -174.06 ry -29.54 rz -11.91 deg; joints [8.488, -43.079, 98.424, -73.976, 64.222, 145.834]
  MoveL 305 to (-206.05, 300.83, -11.57) mm, rotated rx -174.06 ry -29.54 rz -11.91 deg; joints [8.274, -42.97, 98.51, -74.227, 64.051, 146.006]
  MoveL 306 to (-201.08, 300.83, -20.25) mm, rotated rx -174.06 ry -29.54 rz -11.91 deg; joints [8.457, -42.524, 98.439, -74.265, 64.049, 146.438]
  MoveL 307 to (-201.08, 297.66, -20.25) mm, rotated rx -174.06 ry -29.54 rz -11.91 deg; joints [8.474, -42.673, 98.745, -74.325, 64.016, 146.609]
  MoveL 308 to (-206.05, 297.66, -11.57) mm, rotated rx -174.06 ry -29.54 rz -11.91 deg; joints [8.291, -43.121, 98.816, -74.287, 64.018, 146.175]
  MoveL 309 to (-200.15, 297.66, -8.41) mm, rotated rx -174.06 ry -29.54 rz -11.91 deg; joints [8.505, -43.23, 98.73, -74.035, 64.188, 146.003]
  MoveL 310 to (-197.85, 297.66, -8.4) mm, rotated rx -174.06 ry -29.54 rz -11.91 deg; joints [8.589, -43.214, 98.696, -73.963, 64.239, 145.998]
  MoveL 311 to (-197.85, 297.66, -4.14) mm, rotated rx -174.06 ry -29.54 rz -11.91 deg; joints [8.588, -43.416, 98.693, -73.869, 64.295, 145.779]
  Set speed (38.1 mm/s)
  MoveL 312 to (-197.89, 297.66, -3.98) mm, rotated rx -174.06 ry -29.54 rz -11.91 deg; joints [8.587, -43.424, 98.694, -73.867, 64.297, 145.771]
  MoveL 313 to (-198.05, 297.34, -3.7) mm, rotated rx -174.06 ry -29.54 rz -11.91 deg; joints [8.583, -43.453, 98.726, -73.872, 64.293, 145.774]
  Set speed (76.2 mm/s)
  MoveL 314 to (-198.05, 294.8, -3.7) mm, rotated rx -174.06 ry -29.54 rz -11.91 deg; joints [8.597, -43.574, 98.971, -73.918, 64.267, 145.908]
  Set speed (38.1 mm/s)
  MoveL 315 to (-197.89, 294.48, -3.98) mm, rotated rx -174.06 ry -29.54 rz -11.91 deg; joints [8.605, -43.575, 98.999, -73.925, 64.263, 145.939]
  MoveL 316 to (-197.85, 294.48, -4.14) mm, rotated rx -174.06 ry -29.54 rz -11.91 deg; joints [8.606, -43.567, 98.998, -73.927, 64.262, 145.947]
  Set speed (76.2 mm/s)
  MoveL 317 to (-197.85, 294.48, -8.4) mm, rotated rx -174.06 ry -29.54 rz -11.91 deg; joints [8.607, -43.365, 99.002, -74.022, 64.206, 146.166]
  MoveL 318 to (-200.15, 294.48, -8.41) mm, rotated rx -174.06 ry -29.54 rz -11.91 deg; joints [8.523, -43.381, 99.035, -74.094, 64.155, 146.171]
  MoveL 319 to (-206.05, 294.48, -11.57) mm, rotated rx -174.06 ry -29.54 rz -11.91 deg; joints [8.308, -43.271, 99.122, -74.347, 63.986, 146.344]
  MoveL 320 to (-201.08, 294.48, -20.25) mm, rotated rx -174.06 ry -29.54 rz -11.91 deg; joints [8.492, -42.822, 99.05, -74.385, 63.983, 146.779]
  MoveL 321 to (-201.08, 291.31, -20.25) mm, rotated rx -174.06 ry -29.54 rz -11.91 deg; joints [8.509, -42.971, 99.355, -74.445, 63.951, 146.949]
  MoveL 322 to (-206.05, 291.31, -11.57) mm, rotated rx -174.06 ry -29.54 rz -11.91 deg; joints [8.325, -43.421, 99.426, -74.407, 63.953, 146.513]
  MoveL 323 to (-200.15, 291.31, -8.41) mm, rotated rx -174.06 ry -29.54 rz -11.91 deg; joints [8.54, -43.531, 99.34, -74.152, 64.123, 146.339]
  MoveL 324 to (-197.85, 291.31, -8.4) mm, rotated rx -174.06 ry -29.54 rz -11.91 deg; joints [8.625, -43.515, 99.306, -74.08, 64.173, 146.334]
  MoveL 325 to (-197.85, 291.31, -4.14) mm, rotated rx -174.06 ry -29.54 rz -11.91 deg; joints [8.624, -43.718, 99.303, -73.985, 64.229, 146.114]
  Set speed (38.1 mm/s)
  MoveL 326 to (-197.89, 291.31, -3.98) mm, rotated rx -174.06 ry -29.54 rz -11.91 deg; joints [8.622, -43.726, 99.304, -73.983, 64.231, 146.106]
  MoveL 327 to (-198.05, 290.99, -3.7) mm, rotated rx -174.06 ry -29.54 rz -11.91 deg; joints [8.618, -43.755, 99.336, -73.988, 64.227, 146.109]
  Set speed (76.2 mm/s)
  MoveL 328 to (-198.05, 288.45, -3.7) mm, rotated rx -174.06 ry -29.54 rz -11.91 deg; joints [8.633, -43.875, 99.579, -74.034, 64.201, 146.242]
  Set speed (38.1 mm/s)
  MoveL 329 to (-197.89, 288.13, -3.98) mm, rotated rx -174.06 ry -29.54 rz -11.91 deg; joints [8.64, -43.876, 99.607, -74.041, 64.198, 146.273]
  MoveL 330 to (-197.85, 288.13, -4.14) mm, rotated rx -174.06 ry -29.54 rz -11.91 deg; joints [8.642, -43.868, 99.607, -74.043, 64.197, 146.281]
  Set speed (76.2 mm/s)
  MoveL 331 to (-197.85, 288.13, -8.4) mm, rotated rx -174.06 ry -29.54 rz -11.91 deg; joints [8.643, -43.665, 99.61, -74.139, 64.141, 146.502]
  MoveL 332 to (-200.15, 288.13, -8.41) mm, rotated rx -174.06 ry -29.54 rz -11.91 deg; joints [8.558, -43.681, 99.644, -74.211, 64.09, 146.506]
  MoveL 333 to (-206.05, 288.13, -11.57) mm, rotated rx -174.06 ry -29.54 rz -11.91 deg; joints [8.342, -43.57, 99.73, -74.467, 63.921, 146.681]
  MoveL 334 to (-201.08, 288.13, -20.25) mm, rotated rx -174.06 ry -29.54 rz -11.91 deg; joints [8.527, -43.12, 99.658, -74.505, 63.918, 147.118]
  MoveL 335 to (-201.08, 284.96, -20.25) mm, rotated rx -174.06 ry -29.54 rz -11.91 deg; joints [8.545, -43.267, 99.961, -74.565, 63.886, 147.288]
  MoveL 336 to (-206.05, 284.96, -11.57) mm, rotated rx -174.06 ry -29.54 rz -11.91 deg; joints [8.36, -43.719, 100.033, -74.526, 63.889, 146.849]
  MoveL 337 to (-200.15, 284.96, -8.41) mm, rotated rx -174.06 ry -29.54 rz -11.91 deg; joints [8.576, -43.83, 99.947, -74.269, 64.058, 146.674]
  MoveL 338 to (-197.85, 284.96, -8.4) mm, rotated rx -174.06 ry -29.54 rz -11.91 deg; joints [8.661, -43.815, 99.913, -74.197, 64.109, 146.669]
  MoveL 339 to (-197.85, 284.96, -4.14) mm, rotated rx -174.06 ry -29.54 rz -11.91 deg; joints [8.66, -44.018, 99.91, -74.101, 64.165, 146.447]
  Set speed (38.1 mm/s)
  MoveL 340 to (-197.89, 284.96, -3.98) mm, rotated rx -174.06 ry -29.54 rz -11.91 deg; joints [8.658, -44.026, 99.91, -74.099, 64.166, 146.439]
  MoveL 341 to (-198.05, 284.64, -3.7) mm, rotated rx -174.06 ry -29.54 rz -11.91 deg; joints [8.654, -44.055, 99.943, -74.103, 64.163, 146.442]
  Set speed (76.2 mm/s)
  MoveL 342 to (-198.05, 282.1, -3.7) mm, rotated rx -174.06 ry -29.54 rz -11.91 deg; joints [8.668, -44.175, 100.184, -74.149, 64.137, 146.575]
  Set speed (38.1 mm/s)
  MoveL 343 to (-197.89, 281.78, -3.98) mm, rotated rx -174.06 ry -29.54 rz -11.91 deg; joints [8.676, -44.176, 100.212, -74.156, 64.134, 146.605]
  MoveL 344 to (-197.85, 281.78, -4.14) mm, rotated rx -174.06 ry -29.54 rz -11.91 deg; joints [8.678, -44.168, 100.212, -74.159, 64.133, 146.614]
  Set speed (76.2 mm/s)
  MoveL 345 to (-197.85, 281.78, -8.4) mm, rotated rx -174.06 ry -29.54 rz -11.91 deg; joints [8.679, -43.964, 100.215, -74.255, 64.077, 146.836]
  MoveL 346 to (-200.15, 281.78, -8.41) mm, rotated rx -174.06 ry -29.54 rz -11.91 deg; joints [8.594, -43.979, 100.249, -74.328, 64.026, 146.841]
  MoveL 347 to (-206.05, 281.78, -11.57) mm, rotated rx -174.06 ry -29.54 rz -11.91 deg; joints [8.377, -43.868, 100.335, -74.585, 63.858, 147.017]
  MoveL 348 to (-201.08, 281.78, -20.25) mm, rotated rx -174.06 ry -29.54 rz -11.91 deg; joints [8.562, -43.415, 100.263, -74.624, 63.855, 147.457]
  MoveL 349 to (-201.08, 278.61, -20.25) mm, rotated rx -174.06 ry -29.54 rz -11.91 deg; joints [8.58, -43.562, 100.565, -74.684, 63.823, 147.625]
  MoveL 350 to (-206.05, 278.61, -11.57) mm, rotated rx -174.06 ry -29.54 rz -11.91 deg; joints [8.395, -44.016, 100.636, -74.645, 63.826, 147.184]
  MoveL 351 to (-200.15, 278.61, -8.41) mm, rotated rx -174.06 ry -29.54 rz -11.91 deg; joints [8.612, -44.128, 100.55, -74.386, 63.995, 147.007]
  MoveL 352 to (-197.85, 278.61, -8.4) mm, rotated rx -174.06 ry -29.54 rz -11.91 deg; joints [8.697, -44.112, 100.516, -74.312, 64.045, 147.002]
  MoveL 353 to (-197.85, 278.61, -4.14) mm, rotated rx -174.06 ry -29.54 rz -11.91 deg; joints [8.696, -44.317, 100.513, -74.216, 64.101, 146.779]
  Set speed (38.1 mm/s)
  MoveL 354 to (-197.89, 278.61, -3.98) mm, rotated rx -174.06 ry -29.54 rz -11.91 deg; joints [8.694, -44.325, 100.514, -74.214, 64.102, 146.771]
  MoveL 355 to (-198.05, 278.29, -3.7) mm, rotated rx -174.06 ry -29.54 rz -11.91 deg; joints [8.69, -44.354, 100.546, -74.218, 64.099, 146.774]
  Set speed (76.2 mm/s)
  MoveL 356 to (-198.05, 275.75, -3.7) mm, rotated rx -174.06 ry -29.54 rz -11.91 deg; joints [8.705, -44.473, 100.786, -74.264, 64.074, 146.906]
  Set speed (38.1 mm/s)
  MoveL 357 to (-197.89, 275.43, -3.98) mm, rotated rx -174.06 ry -29.54 rz -11.91 deg; joints [8.712, -44.474, 100.814, -74.271, 64.07, 146.937]
  MoveL 358 to (-197.85, 275.43, -4.14) mm, rotated rx -174.06 ry -29.54 rz -11.91 deg; joints [8.714, -44.466, 100.814, -74.273, 64.069, 146.945]
  Set speed (76.2 mm/s)
  MoveL 359 to (-197.85, 275.43, -8.4) mm, rotated rx -174.06 ry -29.54 rz -11.91 deg; joints [8.715, -44.261, 100.817, -74.37, 64.013, 147.168]
  MoveL 360 to (-200.15, 275.43, -8.41) mm, rotated rx -174.06 ry -29.54 rz -11.91 deg; joints [8.63, -44.276, 100.851, -74.444, 63.963, 147.173]
  MoveL 361 to (-206.05, 275.43, -11.57) mm, rotated rx -174.06 ry -29.54 rz -11.91 deg; joints [8.412, -44.164, 100.937, -74.704, 63.795, 147.351]
  MoveL 362 to (-201.08, 275.43, -20.25) mm, rotated rx -174.06 ry -29.54 rz -11.91 deg; joints [8.598, -43.709, 100.865, -74.743, 63.792, 147.793]
  MoveL 363 to (-201.08, 272.26, -20.25) mm, rotated rx -174.06 ry -29.54 rz -11.91 deg; joints [8.616, -43.855, 101.165, -74.802, 63.761, 147.961]
  MoveL 364 to (-206.05, 272.26, -11.57) mm, rotated rx -174.06 ry -29.54 rz -11.91 deg; joints [8.43, -44.311, 101.236, -74.762, 63.765, 147.518]
  MoveL 365 to (-200.15, 272.26, -8.41) mm, rotated rx -174.06 ry -29.54 rz -11.91 deg; joints [8.648, -44.424, 101.15, -74.501, 63.932, 147.339]
  MoveL 366 to (-197.85, 272.26, -8.4) mm, rotated rx -174.06 ry -29.54 rz -11.91 deg; joints [8.733, -44.408, 101.117, -74.428, 63.982, 147.334]
  MoveL 367 to (-197.85, 272.26, -4.14) mm, rotated rx -174.06 ry -29.54 rz -11.91 deg; joints [8.732, -44.614, 101.113, -74.33, 64.038, 147.11]
  Set speed (38.1 mm/s)
  MoveL 368 to (-197.89, 272.26, -3.98) mm, rotated rx -174.06 ry -29.54 rz -11.91 deg; joints [8.731, -44.622, 101.114, -74.328, 64.039, 147.102]
  MoveL 369 to (-198.05, 271.94, -3.7) mm, rotated rx -174.06 ry -29.54 rz -11.91 deg; joints [8.726, -44.651, 101.146, -74.332, 64.036, 147.104]
  Set speed (76.2 mm/s)
  MoveL 370 to (-198.05, 269.4, -3.7) mm, rotated rx -174.06 ry -29.54 rz -11.91 deg; joints [8.741, -44.77, 101.385, -74.378, 64.011, 147.236]
  Set speed (38.1 mm/s)
  MoveL 371 to (-197.89, 269.08, -3.98) mm, rotated rx -174.06 ry -29.54 rz -11.91 deg; joints [8.749, -44.77, 101.413, -74.385, 64.008, 147.266]
  MoveL 372 to (-197.85, 269.08, -4.14) mm, rotated rx -174.06 ry -29.54 rz -11.91 deg; joints [8.75, -44.762, 101.412, -74.387, 64.007, 147.275]
  Set speed (76.2 mm/s)
  MoveL 373 to (-197.85, 269.08, -8.4) mm, rotated rx -174.06 ry -29.54 rz -11.91 deg; joints [8.751, -44.556, 101.416, -74.485, 63.951, 147.499]
  MoveL 374 to (-200.15, 269.08, -8.41) mm, rotated rx -174.06 ry -29.54 rz -11.91 deg; joints [8.666, -44.571, 101.449, -74.559, 63.901, 147.505]
  MoveL 375 to (-206.05, 269.08, -11.57) mm, rotated rx -174.06 ry -29.54 rz -11.91 deg; joints [8.447, -44.458, 101.535, -74.821, 63.734, 147.684]
  MoveL 376 to (-201.08, 269.08, -20.25) mm, rotated rx -174.06 ry -29.54 rz -11.91 deg; joints [8.634, -44.001, 101.464, -74.861, 63.731, 148.129]
  MoveL 377 to (-201.08, 265.91, -20.25) mm, rotated rx -174.06 ry -29.54 rz -11.91 deg; joints [8.652, -44.146, 101.762, -74.92, 63.7, 148.296]
  MoveL 378 to (-206.05, 265.91, -11.57) mm, rotated rx -174.06 ry -29.54 rz -11.91 deg; joints [8.465, -44.604, 101.833, -74.88, 63.704, 147.85]
  MoveL 379 to (-200.15, 265.91, -8.41) mm, rotated rx -174.06 ry -29.54 rz -11.91 deg; joints [8.684, -44.718, 101.747, -74.616, 63.871, 147.67]
  MoveL 380 to (-197.85, 265.91, -8.4) mm, rotated rx -174.06 ry -29.54 rz -11.91 deg; joints [8.77, -44.703, 101.714, -74.542, 63.921, 147.665]
  MoveL 381 to (-197.85, 265.91, -4.14) mm, rotated rx -174.06 ry -29.54 rz -11.91 deg; joints [8.769, -44.91, 101.711, -74.444, 63.976, 147.439]
  Set speed (38.1 mm/s)
  MoveL 382 to (-197.89, 265.91, -3.98) mm, rotated rx -174.06 ry -29.54 rz -11.91 deg; joints [8.767, -44.918, 101.711, -74.442, 63.977, 147.431]
  MoveL 383 to (-198.05, 265.59, -3.7) mm, rotated rx -174.06 ry -29.54 rz -11.91 deg; joints [8.763, -44.947, 101.743, -74.446, 63.975, 147.433]
  Set speed (76.2 mm/s)
  MoveL 384 to (-198.05, 263.05, -3.7) mm, rotated rx -174.06 ry -29.54 rz -11.91 deg; joints [8.778, -45.065, 101.981, -74.491, 63.95, 147.564]
  Set speed (38.1 mm/s)
  MoveL 385 to (-197.89, 262.73, -3.98) mm, rotated rx -174.06 ry -29.54 rz -11.91 deg; joints [8.786, -45.065, 102.008, -74.498, 63.947, 147.595]
  MoveL 386 to (-197.85, 262.73, -4.14) mm, rotated rx -174.06 ry -29.54 rz -11.91 deg; joints [8.787, -45.057, 102.008, -74.5, 63.946, 147.603]
  Set speed (76.2 mm/s)
  MoveL 387 to (-197.85, 262.73, -8.4) mm, rotated rx -174.06 ry -29.54 rz -11.91 deg; joints [8.788, -44.849, 102.011, -74.599, 63.89, 147.829]
  MoveL 388 to (-200.15, 262.73, -8.41) mm, rotated rx -174.06 ry -29.54 rz -11.91 deg; joints [8.702, -44.865, 102.045, -74.674, 63.84, 147.835]
  MoveL 389 to (-206.05, 262.73, -11.57) mm, rotated rx -174.06 ry -29.54 rz -11.91 deg; joints [8.483, -44.751, 102.131, -74.938, 63.674, 148.016]
  MoveL 390 to (-201.08, 262.73, -20.25) mm, rotated rx -174.06 ry -29.54 rz -11.91 deg; joints [8.67, -44.291, 102.059, -74.978, 63.67, 148.463]
  MoveL 391 to (-201.08, 259.56, -20.25) mm, rotated rx -174.06 ry -29.54 rz -11.91 deg; joints [8.689, -44.436, 102.356, -75.037, 63.64, 148.63]
  MoveL 392 to (-206.05, 259.56, -11.57) mm, rotated rx -174.06 ry -29.54 rz -11.91 deg; joints [8.501, -44.896, 102.427, -74.996, 63.644, 148.181]
  MoveL 393 to (-200.15, 259.56, -8.41) mm, rotated rx -174.06 ry -29.54 rz -11.91 deg; joints [8.721, -45.011, 102.341, -74.731, 63.81, 147.999]
  MoveL 394 to (-197.85, 259.56, -8.4) mm, rotated rx -174.06 ry -29.54 rz -11.91 deg; joints [8.807, -44.996, 102.308, -74.656, 63.86, 147.994]
  MoveL 395 to (-197.85, 259.56, -4.14) mm, rotated rx -174.06 ry -29.54 rz -11.91 deg; joints [8.806, -45.204, 102.305, -74.557, 63.916, 147.767]
  Set speed (38.1 mm/s)
  MoveL 396 to (-197.89, 259.56, -3.98) mm, rotated rx -174.06 ry -29.54 rz -11.91 deg; joints [8.804, -45.212, 102.305, -74.554, 63.917, 147.758]
  MoveL 397 to (-198.05, 259.24, -3.7) mm, rotated rx -174.06 ry -29.54 rz -11.91 deg; joints [8.8, -45.241, 102.337, -74.559, 63.914, 147.761]
  Set speed (76.2 mm/s)
  MoveL 398 to (-198.05, 256.7, -3.7) mm, rotated rx -174.06 ry -29.54 rz -11.91 deg; joints [8.815, -45.358, 102.574, -74.604, 63.89, 147.891]
  Set speed (38.1 mm/s)
  MoveL 399 to (-197.89, 256.38, -3.98) mm, rotated rx -174.06 ry -29.54 rz -11.91 deg; joints [8.823, -45.358, 102.601, -74.611, 63.887, 147.922]
  MoveL 400 to (-197.85, 256.38, -4.14) mm, rotated rx -174.06 ry -29.54 rz -11.91 deg; joints [8.824, -45.35, 102.601, -74.613, 63.886, 147.93]
  Set speed (76.2 mm/s)
  MoveL 401 to (-197.85, 256.38, -8.4) mm, rotated rx -174.06 ry -29.54 rz -11.91 deg; joints [8.825, -45.142, 102.604, -74.713, 63.83, 148.158]
  MoveL 402 to (-200.15, 256.38, -8.41) mm, rotated rx -174.06 ry -29.54 rz -11.91 deg; joints [8.739, -45.157, 102.637, -74.788, 63.78, 148.164]
  MoveL 403 to (-206.05, 256.38, -11.57) mm, rotated rx -174.06 ry -29.54 rz -11.91 deg; joints [8.519, -45.042, 102.723, -75.054, 63.614, 148.346]
  MoveL 404 to (-201.08, 256.38, -20.25) mm, rotated rx -174.06 ry -29.54 rz -11.91 deg; joints [8.707, -44.58, 102.652, -75.095, 63.61, 148.796]
  MoveL 405 to (-201.08, 253.21, -20.25) mm, rotated rx -174.06 ry -29.54 rz -11.91 deg; joints [8.726, -44.724, 102.947, -75.153, 63.581, 148.962]
  MoveL 406 to (-206.05, 253.21, -11.57) mm, rotated rx -174.06 ry -29.54 rz -11.91 deg; joints [8.537, -45.187, 103.018, -75.112, 63.585, 148.51]
  MoveL 407 to (-200.15, 253.21, -8.41) mm, rotated rx -174.06 ry -29.54 rz -11.91 deg; joints [8.757, -45.303, 102.933, -74.845, 63.751, 148.328]
  MoveL 408 to (-197.85, 253.21, -8.4) mm, rotated rx -174.06 ry -29.54 rz -11.91 deg; joints [8.844, -45.287, 102.899, -74.769, 63.8, 148.322]
  MoveL 409 to (-197.85, 253.21, -4.14) mm, rotated rx -174.06 ry -29.54 rz -11.91 deg; joints [8.843, -45.496, 102.896, -74.669, 63.856, 148.093]
  Set speed (38.1 mm/s)
  MoveL 410 to (-197.89, 253.21, -3.98) mm, rotated rx -174.06 ry -29.54 rz -11.91 deg; joints [8.841, -45.504, 102.896, -74.667, 63.857, 148.085]
  MoveL 411 to (-198.05, 252.89, -3.7) mm, rotated rx -174.06 ry -29.54 rz -11.91 deg; joints [8.837, -45.533, 102.928, -74.671, 63.854, 148.087]
  Set speed (76.2 mm/s)
  MoveL 412 to (-198.05, 250.35, -3.7) mm, rotated rx -174.06 ry -29.54 rz -11.91 deg; joints [8.852, -45.65, 103.163, -74.716, 63.831, 148.217]
  Set speed (38.1 mm/s)
  MoveL 413 to (-197.89, 250.03, -3.98) mm, rotated rx -174.06 ry -29.54 rz -11.91 deg; joints [8.86, -45.65, 103.191, -74.723, 63.827, 148.248]
  MoveL 414 to (-197.85, 250.03, -4.14) mm, rotated rx -174.06 ry -29.54 rz -11.91 deg; joints [8.862, -45.642, 103.19, -74.725, 63.826, 148.256]
  Set speed (76.2 mm/s)
  MoveL 415 to (-197.85, 250.03, -8.4) mm, rotated rx -174.06 ry -29.54 rz -11.91 deg; joints [8.863, -45.432, 103.193, -74.825, 63.771, 148.485]
  MoveL 416 to (-200.15, 250.03, -8.41) mm, rotated rx -174.06 ry -29.54 rz -11.91 deg; joints [8.776, -45.448, 103.227, -74.901, 63.721, 148.491]
  MoveL 417 to (-206.05, 250.03, -11.57) mm, rotated rx -174.06 ry -29.54 rz -11.91 deg; joints [8.555, -45.332, 103.312, -75.17, 63.556, 148.675]
  MoveL 418 to (-201.08, 250.03, -20.25) mm, rotated rx -174.06 ry -29.54 rz -11.91 deg; joints [8.744, -44.868, 103.242, -75.211, 63.552, 149.127]
  MoveL 419 to (-201.08, 246.86, -20.25) mm, rotated rx -174.06 ry -29.54 rz -11.91 deg; joints [8.763, -45.011, 103.535, -75.269, 63.523, 149.293]
  MoveL 420 to (-206.05, 246.86, -11.57) mm, rotated rx -174.06 ry -29.54 rz -11.91 deg; joints [8.573, -45.476, 103.606, -75.228, 63.527, 148.839]
  MoveL 421 to (-200.15, 246.86, -8.41) mm, rotated rx -174.06 ry -29.54 rz -11.91 deg; joints [8.795, -45.593, 103.521, -74.958, 63.692, 148.654]
  MoveL 422 to (-197.85, 246.86, -8.4) mm, rotated rx -174.06 ry -29.54 rz -11.91 deg; joints [8.882, -45.577, 103.487, -74.882, 63.742, 148.648]
  MoveL 423 to (-197.85, 246.86, -4.14) mm, rotated rx -174.06 ry -29.54 rz -11.91 deg; joints [8.881, -45.787, 103.484, -74.781, 63.797, 148.419]
  Set speed (38.1 mm/s)
  MoveL 424 to (-197.89, 246.86, -3.98) mm, rotated rx -174.06 ry -29.54 rz -11.91 deg; joints [8.879, -45.795, 103.484, -74.779, 63.798, 148.41]
  MoveL 425 to (-198.05, 246.54, -3.7) mm, rotated rx -174.06 ry -29.54 rz -11.91 deg; joints [8.875, -45.825, 103.516, -74.783, 63.795, 148.412]
  Set speed (76.2 mm/s)
  MoveL 426 to (-198.05, 244, -3.7) mm, rotated rx -174.06 ry -29.54 rz -11.91 deg; joints [8.89, -45.941, 103.75, -74.827, 63.772, 148.542]
  Set speed (38.1 mm/s)
  MoveL 427 to (-197.89, 243.69, -3.98) mm, rotated rx -174.06 ry -29.54 rz -11.91 deg; joints [8.898, -45.94, 103.777, -74.834, 63.769, 148.572]
  MoveL 428 to (-197.85, 243.69, -4.14) mm, rotated rx -174.06 ry -29.54 rz -11.91 deg; joints [8.9, -45.932, 103.777, -74.837, 63.768, 148.581]
  Set speed (76.2 mm/s)
  MoveL 429 to (-197.85, 243.69, -8.4) mm, rotated rx -174.06 ry -29.54 rz -11.91 deg; joints [8.901, -45.721, 103.78, -74.938, 63.713, 148.811]
  MoveL 430 to (-200.15, 243.69, -8.41) mm, rotated rx -174.06 ry -29.54 rz -11.91 deg; joints [8.813, -45.737, 103.814, -75.014, 63.663, 148.817]
  MoveL 431 to (-206.05, 243.69, -11.57) mm, rotated rx -174.06 ry -29.54 rz -11.91 deg; joints [8.592, -45.62, 103.899, -75.285, 63.498, 149.003]
  MoveL 432 to (-201.08, 243.69, -20.25) mm, rotated rx -174.06 ry -29.54 rz -11.91 deg; joints [8.781, -45.154, 103.828, -75.327, 63.494, 149.458]
  MoveL 433 to (-201.08, 240.51, -20.25) mm, rotated rx -174.06 ry -29.54 rz -11.91 deg; joints [8.8, -45.296, 104.12, -75.384, 63.466, 149.623]
  MoveL 434 to (-206.05, 240.51, -11.57) mm, rotated rx -174.06 ry -29.54 rz -11.91 deg; joints [8.61, -45.763, 104.191, -75.343, 63.47, 149.166]
  MoveL 435 to (-200.15, 240.51, -8.41) mm, rotated rx -174.06 ry -29.54 rz -11.91 deg; joints [8.832, -45.881, 104.106, -75.071, 63.635, 148.98]
  MoveL 436 to (-197.85, 240.51, -8.4) mm, rotated rx -174.06 ry -29.54 rz -11.91 deg; joints [8.92, -45.866, 104.072, -74.994, 63.684, 148.974]
  MoveL 437 to (-197.85, 240.51, -4.14) mm, rotated rx -174.06 ry -29.54 rz -11.91 deg; joints [8.919, -46.077, 104.069, -74.892, 63.739, 148.743]
  Set speed (38.1 mm/s)
  MoveL 438 to (-197.89, 240.51, -3.98) mm, rotated rx -174.06 ry -29.54 rz -11.91 deg; joints [8.917, -46.085, 104.07, -74.89, 63.74, 148.734]
  MoveL 439 to (-198.05, 240.19, -3.7) mm, rotated rx -174.06 ry -29.54 rz -11.91 deg; joints [8.913, -46.114, 104.101, -74.894, 63.738, 148.736]
  Set speed (76.2 mm/s)
  MoveL 440 to (-198.05, 237.65, -3.7) mm, rotated rx -174.06 ry -29.54 rz -11.91 deg; joints [8.928, -46.23, 104.334, -74.938, 63.715, 148.865]
  Set speed (38.1 mm/s)
  MoveL 441 to (-197.89, 237.34, -3.98) mm, rotated rx -174.06 ry -29.54 rz -11.91 deg; joints [8.936, -46.229, 104.361, -74.945, 63.712, 148.895]
  MoveL 442 to (-197.85, 237.34, -4.14) mm, rotated rx -174.06 ry -29.54 rz -11.91 deg; joints [8.938, -46.221, 104.361, -74.947, 63.711, 148.904]
  Set speed (76.2 mm/s)
  MoveL 443 to (-197.85, 237.34, -8.4) mm, rotated rx -174.06 ry -29.54 rz -11.91 deg; joints [8.939, -46.009, 104.364, -75.049, 63.655, 149.136]
  MoveL 444 to (-200.15, 237.34, -8.41) mm, rotated rx -174.06 ry -29.54 rz -11.91 deg; joints [8.851, -46.025, 104.397, -75.127, 63.606, 149.142]
  MoveL 445 to (-206.05, 237.34, -11.57) mm, rotated rx -174.06 ry -29.54 rz -11.91 deg; joints [8.628, -45.907, 104.483, -75.4, 63.442, 149.329]
  MoveL 446 to (-201.08, 237.34, -20.25) mm, rotated rx -174.06 ry -29.54 rz -11.91 deg; joints [8.819, -45.438, 104.412, -75.442, 63.437, 149.787]
  MoveL 447 to (-201.08, 234.16, -20.25) mm, rotated rx -174.06 ry -29.54 rz -11.91 deg; joints [8.838, -45.58, 104.703, -75.499, 63.409, 149.951]
  MoveL 448 to (-206.05, 234.16, -11.57) mm, rotated rx -174.06 ry -29.54 rz -11.91 deg; joints [8.647, -46.05, 104.774, -75.457, 63.414, 149.492]
  MoveL 449 to (-200.15, 234.16, -8.41) mm, rotated rx -174.06 ry -29.54 rz -11.91 deg; joints [8.87, -46.168, 104.688, -75.182, 63.578, 149.304]
  MoveL 450 to (-197.85, 234.16, -8.4) mm, rotated rx -174.06 ry -29.54 rz -11.91 deg; joints [8.958, -46.153, 104.655, -75.105, 63.627, 149.298]
  MoveL 451 to (-197.85, 234.16, -4.14) mm, rotated rx -174.06 ry -29.54 rz -11.91 deg; joints [8.957, -46.365, 104.651, -75.003, 63.682, 149.065]
  Set speed (38.1 mm/s)
  MoveL 452 to (-197.89, 234.16, -3.98) mm, rotated rx -174.06 ry -29.54 rz -11.91 deg; joints [8.955, -46.373, 104.652, -75, 63.683, 149.057]
  MoveL 453 to (-198.05, 233.84, -3.7) mm, rotated rx -174.06 ry -29.54 rz -11.91 deg; joints [8.951, -46.402, 104.683, -75.004, 63.681, 149.058]
  Set speed (76.2 mm/s)
  MoveL 454 to (-198.05, 231.3, -3.7) mm, rotated rx -174.06 ry -29.54 rz -11.91 deg; joints [8.966, -46.517, 104.915, -75.048, 63.658, 149.187]
  Set speed (38.1 mm/s)
  MoveL 455 to (-197.89, 230.99, -3.98) mm, rotated rx -174.06 ry -29.54 rz -11.91 deg; joints [8.974, -46.517, 104.942, -75.055, 63.655, 149.218]
  MoveL 456 to (-197.85, 230.99, -4.14) mm, rotated rx -174.06 ry -29.54 rz -11.91 deg; joints [8.976, -46.509, 104.942, -75.058, 63.654, 149.226]
  Set speed (76.2 mm/s)
  MoveL 457 to (-197.85, 230.99, -8.4) mm, rotated rx -174.06 ry -29.54 rz -11.91 deg; joints [8.977, -46.296, 104.945, -75.16, 63.599, 149.46]
  MoveL 458 to (-200.15, 230.99, -8.41) mm, rotated rx -174.06 ry -29.54 rz -11.91 deg; joints [8.889, -46.311, 104.978, -75.238, 63.55, 149.466]
  MoveL 459 to (-206.05, 230.99, -11.57) mm, rotated rx -174.06 ry -29.54 rz -11.91 deg; joints [8.665, -46.192, 105.064, -75.514, 63.386, 149.654]
  MoveL 460 to (-201.08, 230.99, -20.25) mm, rotated rx -174.06 ry -29.54 rz -11.91 deg; joints [8.857, -45.721, 104.993, -75.556, 63.382, 150.115]
  MoveL 461 to (-201.08, 227.81, -20.25) mm, rotated rx -174.06 ry -29.54 rz -11.91 deg; joints [8.876, -45.862, 105.282, -75.613, 63.354, 150.279]
  MoveL 462 to (-206.05, 227.81, -11.57) mm, rotated rx -174.06 ry -29.54 rz -11.91 deg; joints [8.684, -46.334, 105.353, -75.57, 63.359, 149.817]
  MoveL 463 to (-200.15, 227.81, -8.41) mm, rotated rx -174.06 ry -29.54 rz -11.91 deg; joints [8.908, -46.454, 105.268, -75.294, 63.522, 149.628]
  MoveL 464 to (-197.85, 227.81, -8.4) mm, rotated rx -174.06 ry -29.54 rz -11.91 deg; joints [8.996, -46.438, 105.234, -75.216, 63.571, 149.621]
  MoveL 465 to (-197.85, 227.81, -4.14) mm, rotated rx -174.06 ry -29.54 rz -11.91 deg; joints [8.995, -46.652, 105.231, -75.112, 63.626, 149.387]
  Set speed (38.1 mm/s)
  MoveL 466 to (-197.89, 227.81, -3.98) mm, rotated rx -174.06 ry -29.54 rz -11.91 deg; joints [8.994, -46.66, 105.232, -75.11, 63.627, 149.378]
  MoveL 467 to (-198.05, 227.49, -3.7) mm, rotated rx -174.06 ry -29.54 rz -11.91 deg; joints [8.989, -46.689, 105.262, -75.114, 63.625, 149.379]
  Set speed (76.2 mm/s)
  MoveL 468 to (-198.05, 224.95, -3.7) mm, rotated rx -174.06 ry -29.54 rz -11.91 deg; joints [9.005, -46.804, 105.494, -75.158, 63.603, 149.508]
  Set speed (38.1 mm/s)
  MoveL 469 to (-197.89, 224.64, -3.98) mm, rotated rx -174.06 ry -29.54 rz -11.91 deg; joints [9.013, -46.803, 105.52, -75.165, 63.6, 149.538]
  MoveL 470 to (-197.85, 224.64, -4.14) mm, rotated rx -174.06 ry -29.54 rz -11.91 deg; joints [9.015, -46.795, 105.52, -75.167, 63.598, 149.547]
  Set speed (76.2 mm/s)
  MoveL 471 to (-197.85, 224.64, -8.4) mm, rotated rx -174.06 ry -29.54 rz -11.91 deg; joints [9.016, -46.58, 105.523, -75.271, 63.543, 149.782]
  MoveL 472 to (-200.15, 224.64, -8.41) mm, rotated rx -174.06 ry -29.54 rz -11.91 deg; joints [8.928, -46.596, 105.557, -75.349, 63.495, 149.789]
  MoveL 473 to (-206.05, 224.64, -11.57) mm, rotated rx -174.06 ry -29.54 rz -11.91 deg; joints [8.703, -46.476, 105.642, -75.627, 63.332, 149.979]
  MoveL 474 to (-201.08, 224.64, -20.25) mm, rotated rx -174.06 ry -29.54 rz -11.91 deg; joints [8.895, -46.003, 105.571, -75.67, 63.327, 150.442]
  MoveL 475 to (-201.08, 221.46, -20.25) mm, rotated rx -174.06 ry -29.54 rz -11.91 deg; joints [8.914, -46.143, 105.859, -75.726, 63.3, 150.605]
  MoveL 476 to (-206.05, 221.46, -11.57) mm, rotated rx -174.06 ry -29.54 rz -11.91 deg; joints [8.722, -46.618, 105.93, -75.683, 63.305, 150.14]
  MoveL 477 to (-200.15, 221.46, -8.41) mm, rotated rx -174.06 ry -29.54 rz -11.91 deg; joints [8.947, -46.738, 105.845, -75.405, 63.468, 149.95]
  MoveL 478 to (-197.85, 221.46, -8.4) mm, rotated rx -174.06 ry -29.54 rz -11.91 deg; joints [9.035, -46.722, 105.811, -75.326, 63.516, 149.943]
  MoveL 479 to (-197.85, 221.46, -4.14) mm, rotated rx -174.06 ry -29.54 rz -11.91 deg; joints [9.034, -46.937, 105.808, -75.222, 63.571, 149.707]
  Set speed (38.1 mm/s)
  MoveL 480 to (-197.89, 221.46, -3.98) mm, rotated rx -174.06 ry -29.54 rz -11.91 deg; joints [9.032, -46.946, 105.808, -75.219, 63.572, 149.698]
  MoveL 481 to (-198.05, 221.14, -3.7) mm, rotated rx -174.06 ry -29.54 rz -11.91 deg; joints [9.028, -46.975, 105.839, -75.223, 63.57, 149.7]
  Set speed (76.2 mm/s)
  MoveL 482 to (-198.05, 218.6, -3.7) mm, rotated rx -174.06 ry -29.54 rz -11.91 deg; joints [9.044, -47.089, 106.069, -75.267, 63.548, 149.827]
  Set speed (38.1 mm/s)
  MoveL 483 to (-197.89, 218.29, -3.98) mm, rotated rx -174.06 ry -29.54 rz -11.91 deg; joints [9.052, -47.088, 106.096, -75.273, 63.545, 149.858]
  MoveL 484 to (-197.85, 218.29, -4.14) mm, rotated rx -174.06 ry -29.54 rz -11.91 deg; joints [9.054, -47.08, 106.095, -75.276, 63.544, 149.867]
  Set speed (76.2 mm/s)
  MoveL 485 to (-197.85, 218.29, -8.4) mm, rotated rx -174.06 ry -29.54 rz -11.91 deg; joints [9.055, -46.864, 106.099, -75.381, 63.489, 150.103]
  MoveL 486 to (-200.15, 218.29, -8.41) mm, rotated rx -174.06 ry -29.54 rz -11.91 deg; joints [8.966, -46.879, 106.132, -75.46, 63.441, 150.11]
  MoveL 487 to (-206.05, 218.29, -11.57) mm, rotated rx -174.06 ry -29.54 rz -11.91 deg; joints [8.741, -46.759, 106.217, -75.74, 63.278, 150.301]
  MoveL 488 to (-201.08, 218.29, -20.25) mm, rotated rx -174.06 ry -29.54 rz -11.91 deg; joints [8.934, -46.283, 106.147, -75.783, 63.273, 150.768]
  MoveL 489 to (-201.08, 215.11, -20.25) mm, rotated rx -174.06 ry -29.54 rz -11.91 deg; joints [8.953, -46.423, 106.433, -75.839, 63.246, 150.93]
  MoveL 490 to (-206.05, 215.11, -11.57) mm, rotated rx -174.06 ry -29.54 rz -11.91 deg; joints [8.76, -46.9, 106.504, -75.796, 63.251, 150.463]
  MoveL 491 to (-200.15, 215.11, -8.41) mm, rotated rx -174.06 ry -29.54 rz -11.91 deg; joints [8.986, -47.021, 106.419, -75.515, 63.414, 150.27]
  MoveL 492 to (-197.85, 215.11, -8.4) mm, rotated rx -174.06 ry -29.54 rz -11.91 deg; joints [9.074, -47.005, 106.385, -75.435, 63.462, 150.264]
  MoveL 493 to (-197.85, 215.11, -4.14) mm, rotated rx -174.06 ry -29.54 rz -11.91 deg; joints [9.073, -47.221, 106.382, -75.33, 63.517, 150.026]
  Set speed (38.1 mm/s)
  MoveL 494 to (-197.89, 215.11, -3.98) mm, rotated rx -174.06 ry -29.54 rz -11.91 deg; joints [9.072, -47.23, 106.383, -75.328, 63.518, 150.017]
  MoveL 495 to (-198.05, 214.79, -3.7) mm, rotated rx -174.06 ry -29.54 rz -11.91 deg; joints [9.067, -47.259, 106.413, -75.332, 63.516, 150.018]
  Set speed (76.2 mm/s)
  MoveL 496 to (-198.05, 212.26, -3.7) mm, rotated rx -174.06 ry -29.54 rz -11.91 deg; joints [9.083, -47.372, 106.642, -75.375, 63.494, 150.146]
  Set speed (38.1 mm/s)
  MoveL 497 to (-197.89, 211.94, -3.98) mm, rotated rx -174.06 ry -29.54 rz -11.91 deg; joints [9.091, -47.371, 106.669, -75.382, 63.491, 150.177]
  MoveL 498 to (-197.85, 211.94, -4.14) mm, rotated rx -174.06 ry -29.54 rz -11.91 deg; joints [9.093, -47.363, 106.668, -75.384, 63.49, 150.185]
  Set speed (76.2 mm/s)
  MoveL 499 to (-197.85, 211.94, -8.4) mm, rotated rx -174.06 ry -29.54 rz -11.91 deg; joints [9.094, -47.146, 106.672, -75.49, 63.435, 150.423]
  MoveL 500 to (-200.15, 211.94, -8.41) mm, rotated rx -174.06 ry -29.54 rz -11.91 deg; joints [9.005, -47.162, 106.705, -75.569, 63.387, 150.43]
  MoveL 501 to (-206.05, 211.94, -11.57) mm, rotated rx -174.06 ry -29.54 rz -11.91 deg; joints [8.779, -47.04, 106.79, -75.852, 63.225, 150.623]
  MoveL 502 to (-201.08, 211.94, -20.25) mm, rotated rx -174.06 ry -29.54 rz -11.91 deg; joints [8.972, -46.562, 106.72, -75.895, 63.22, 151.092]
  MoveL 503 to (-201.08, 208.76, -20.25) mm, rotated rx -174.06 ry -29.54 rz -11.91 deg; joints [8.992, -46.701, 107.005, -75.951, 63.194, 151.254]
  MoveL 504 to (-206.05, 208.76, -11.57) mm, rotated rx -174.06 ry -29.54 rz -11.91 deg; joints [8.798, -47.18, 107.076, -75.907, 63.199, 150.784]
  MoveL 505 to (-200.15, 208.76, -8.41) mm, rotated rx -174.06 ry -29.54 rz -11.91 deg; joints [9.025, -47.302, 106.99, -75.624, 63.361, 150.59]
  MoveL 506 to (-197.85, 208.76, -8.4) mm, rotated rx -174.06 ry -29.54 rz -11.91 deg; joints [9.114, -47.287, 106.957, -75.544, 63.409, 150.583]
  MoveL 507 to (-197.85, 208.76, -4.14) mm, rotated rx -174.06 ry -29.54 rz -11.91 deg; joints [9.113, -47.504, 106.954, -75.438, 63.463, 150.344]
  Set speed (38.1 mm/s)
  MoveL 508 to (-197.89, 208.76, -3.98) mm, rotated rx -174.06 ry -29.54 rz -11.91 deg; joints [9.111, -47.513, 106.954, -75.436, 63.465, 150.335]
  MoveL 509 to (-198.05, 208.45, -3.7) mm, rotated rx -174.06 ry -29.54 rz -11.91 deg; joints [9.107, -47.542, 106.985, -75.44, 63.462, 150.336]
  Set speed (76.2 mm/s)
  MoveL 510 to (-198.05, 205.91, -3.7) mm, rotated rx -174.06 ry -29.54 rz -11.91 deg; joints [9.123, -47.655, 107.213, -75.483, 63.441, 150.463]
  Set speed (38.1 mm/s)
  MoveL 511 to (-197.89, 205.59, -3.98) mm, rotated rx -174.06 ry -29.54 rz -11.91 deg; joints [9.131, -47.654, 107.239, -75.489, 63.438, 150.494]
  MoveL 512 to (-197.85, 205.59, -4.14) mm, rotated rx -174.06 ry -29.54 rz -11.91 deg; joints [9.133, -47.645, 107.239, -75.492, 63.437, 150.503]
  Set speed (76.2 mm/s)
  MoveL 513 to (-197.85, 205.59, -8.4) mm, rotated rx -174.06 ry -29.54 rz -11.91 deg; joints [9.134, -47.427, 107.242, -75.598, 63.382, 150.742]
  MoveL 514 to (-200.15, 205.59, -8.41) mm, rotated rx -174.06 ry -29.54 rz -11.91 deg; joints [9.045, -47.443, 107.275, -75.679, 63.334, 150.75]
  MoveL 515 to (-206.05, 205.59, -11.57) mm, rotated rx -174.06 ry -29.54 rz -11.91 deg; joints [8.817, -47.32, 107.361, -75.963, 63.173, 150.944]
  MoveL 516 to (-201.08, 205.59, -20.25) mm, rotated rx -174.06 ry -29.54 rz -11.91 deg; joints [9.012, -46.839, 107.29, -76.007, 63.168, 151.416]
  MoveL 517 to (-201.08, 202.41, -20.25) mm, rotated rx -174.06 ry -29.54 rz -11.91 deg; joints [9.031, -46.978, 107.574, -76.063, 63.142, 151.577]
  MoveL 518 to (-206.05, 202.41, -11.57) mm, rotated rx -174.06 ry -29.54 rz -11.91 deg; joints [8.836, -47.459, 107.645, -76.018, 63.147, 151.104]
  MoveL 519 to (-200.15, 202.41, -8.41) mm, rotated rx -174.06 ry -29.54 rz -11.91 deg; joints [9.064, -47.583, 107.559, -75.733, 63.308, 150.909]
  MoveL 520 to (-197.85, 202.41, -8.4) mm, rotated rx -174.06 ry -29.54 rz -11.91 deg; joints [9.154, -47.567, 107.526, -75.652, 63.356, 150.902]
  MoveL 521 to (-197.85, 202.41, -4.14) mm, rotated rx -174.06 ry -29.54 rz -11.91 deg; joints [9.153, -47.786, 107.523, -75.545, 63.411, 150.661]
  Set speed (38.1 mm/s)
  MoveL 522 to (-197.89, 202.41, -3.98) mm, rotated rx -174.06 ry -29.54 rz -11.91 deg; joints [9.151, -47.794, 107.523, -75.543, 63.412, 150.652]
  MoveL 523 to (-198.05, 202.1, -3.7) mm, rotated rx -174.06 ry -29.54 rz -11.91 deg; joints [9.147, -47.823, 107.554, -75.547, 63.41, 150.653]
  Set speed (76.2 mm/s)
  MoveL 524 to (-198.05, 199.56, -3.7) mm, rotated rx -174.06 ry -29.54 rz -11.91 deg; joints [9.163, -47.936, 107.78, -75.59, 63.389, 150.779]
  Set speed (38.1 mm/s)
  MoveL 525 to (-197.89, 199.24, -3.98) mm, rotated rx -174.06 ry -29.54 rz -11.91 deg; joints [9.171, -47.934, 107.807, -75.596, 63.386, 150.81]
  MoveL 526 to (-197.85, 199.24, -4.14) mm, rotated rx -174.06 ry -29.54 rz -11.91 deg; joints [9.173, -47.926, 107.806, -75.599, 63.385, 150.819]
  Set speed (76.2 mm/s)
  MoveL 527 to (-197.85, 199.24, -8.4) mm, rotated rx -174.06 ry -29.54 rz -11.91 deg; joints [9.174, -47.707, 107.81, -75.706, 63.33, 151.06]
  MoveL 528 to (-200.15, 199.24, -8.41) mm, rotated rx -174.06 ry -29.54 rz -11.91 deg; joints [9.084, -47.722, 107.843, -75.787, 63.283, 151.068]
  MoveL 529 to (-206.05, 199.24, -11.57) mm, rotated rx -174.06 ry -29.54 rz -11.91 deg; joints [8.856, -47.599, 107.928, -76.074, 63.122, 151.264]
  MoveL 530 to (-201.08, 199.24, -20.25) mm, rotated rx -174.06 ry -29.54 rz -11.91 deg; joints [9.051, -47.116, 107.858, -76.118, 63.116, 151.738]
  MoveL 531 to (-201.08, 196.06, -20.25) mm, rotated rx -174.06 ry -29.54 rz -11.91 deg; joints [9.071, -47.253, 108.14, -76.174, 63.091, 151.899]
  MoveL 532 to (-206.05, 196.06, -11.57) mm, rotated rx -174.06 ry -29.54 rz -11.91 deg; joints [8.875, -47.737, 108.211, -76.129, 63.097, 151.423]
  MoveL 533 to (-200.15, 196.06, -8.41) mm, rotated rx -174.06 ry -29.54 rz -11.91 deg; joints [9.104, -47.861, 108.126, -75.841, 63.257, 151.226]
  MoveL 534 to (-197.85, 196.06, -8.4) mm, rotated rx -174.06 ry -29.54 rz -11.91 deg; joints [9.194, -47.846, 108.092, -75.76, 63.305, 151.219]
  MoveL 535 to (-197.85, 196.06, -4.14) mm, rotated rx -174.06 ry -29.54 rz -11.91 deg; joints [9.193, -48.066, 108.089, -75.652, 63.359, 150.977]
  Set speed (38.1 mm/s)
  MoveL 536 to (-197.89, 196.06, -3.98) mm, rotated rx -174.06 ry -29.54 rz -11.91 deg; joints [9.191, -48.074, 108.09, -75.65, 63.36, 150.968]
  MoveL 537 to (-198.05, 195.75, -3.7) mm, rotated rx -174.06 ry -29.54 rz -11.91 deg; joints [9.187, -48.104, 108.12, -75.653, 63.358, 150.968]
  Set speed (76.2 mm/s)
  MoveL 538 to (-198.05, 193.21, -3.7) mm, rotated rx -174.06 ry -29.54 rz -11.91 deg; joints [9.203, -48.215, 108.346, -75.696, 63.338, 151.094]
  Set speed (38.1 mm/s)
  MoveL 539 to (-197.89, 192.89, -3.98) mm, rotated rx -174.06 ry -29.54 rz -11.91 deg; joints [9.211, -48.214, 108.372, -75.703, 63.335, 151.125]
  MoveL 540 to (-197.85, 192.89, -4.14) mm, rotated rx -174.06 ry -29.54 rz -11.91 deg; joints [9.213, -48.206, 108.371, -75.705, 63.334, 151.134]
  Set speed (76.2 mm/s)
  MoveL 541 to (-197.85, 192.89, -8.4) mm, rotated rx -174.06 ry -29.54 rz -11.91 deg; joints [9.214, -47.985, 108.375, -75.813, 63.279, 151.377]
  MoveL 542 to (-199.6, 192.89, -8.41) mm, rotated rx -174.06 ry -29.54 rz -11.91 deg; joints [9.146, -47.997, 108.4, -75.875, 63.243, 151.383]
  MoveL 543 to (-206.05, 192.89, -11.57) mm, rotated rx -174.06 ry -29.54 rz -11.91 deg; joints [8.895, -47.876, 108.494, -76.184, 63.072, 151.582]
  MoveL 544 to (-201.08, 192.89, -20.25) mm, rotated rx -174.06 ry -29.54 rz -11.91 deg; joints [9.091, -47.39, 108.423, -76.229, 63.066, 152.06]
  MoveL 545 to (-201.08, 189.71, -20.25) mm, rotated rx -174.06 ry -29.54 rz -11.91 deg; joints [9.111, -47.527, 108.704, -76.284, 63.041, 152.22]
  MoveL 546 to (-206.05, 189.71, -11.57) mm, rotated rx -174.06 ry -29.54 rz -11.91 deg; joints [8.914, -48.014, 108.775, -76.239, 63.047, 151.741]
  MoveL 547 to (-199.6, 189.71, -8.41) mm, rotated rx -174.06 ry -29.54 rz -11.91 deg; joints [9.166, -48.135, 108.682, -75.929, 63.218, 151.541]
  MoveL 548 to (-197.85, 189.71, -8.4) mm, rotated rx -174.06 ry -29.54 rz -11.91 deg; joints [9.235, -48.124, 108.656, -75.867, 63.254, 151.535]
  MoveL 549 to (-197.85, 189.71, -4.14) mm, rotated rx -174.06 ry -29.54 rz -11.91 deg; joints [9.233, -48.345, 108.653, -75.758, 63.309, 151.291]
  MoveL 550 to (-197.85, 189.59, -3.66) mm, rotated rx -174.06 ry -29.54 rz -11.91 deg; joints [9.234, -48.375, 108.664, -75.748, 63.314, 151.27]
  MoveL 551 to (-197.85, 189.24, -3.31) mm, rotated rx -174.06 ry -29.54 rz -11.91 deg; joints [9.236, -48.408, 108.695, -75.745, 63.315, 151.268]
  MoveL 552 to (-197.85, 188.76, -3.19) mm, rotated rx -174.06 ry -29.54 rz -11.91 deg; joints [9.239, -48.436, 108.737, -75.75, 63.313, 151.284]
  MoveL 553 to (-197.85, 187.49, -3.19) mm, rotated rx -174.06 ry -29.54 rz -11.91 deg; joints [9.248, -48.492, 108.849, -75.771, 63.303, 151.347]
  MoveL 554 to (-197.85, 187.02, -3.31) mm, rotated rx -174.06 ry -29.54 rz -11.91 deg; joints [9.251, -48.506, 108.891, -75.782, 63.298, 151.377]
  MoveL 555 to (-197.85, 186.67, -3.66) mm, rotated rx -174.06 ry -29.54 rz -11.91 deg; joints [9.253, -48.503, 108.923, -75.797, 63.291, 151.415]
  MoveL 556 to (-197.85, 186.54, -4.14) mm, rotated rx -174.06 ry -29.54 rz -11.91 deg; joints [9.254, -48.484, 108.934, -75.811, 63.283, 151.448]
  MoveL 557 to (-197.85, 186.54, -8.4) mm, rotated rx -174.06 ry -29.54 rz -11.91 deg; joints [9.255, -48.262, 108.938, -75.92, 63.229, 151.693]
  MoveL 558 to (-199.6, 186.54, -8.41) mm, rotated rx -174.06 ry -29.54 rz -11.91 deg; joints [9.186, -48.274, 108.963, -75.982, 63.193, 151.699]
  MoveL 559 to (-206.05, 186.54, -11.57) mm, rotated rx -174.06 ry -29.54 rz -11.91 deg; joints [8.934, -48.152, 109.056, -76.293, 63.022, 151.9]
  MoveL 560 to (-201.08, 186.54, -20.25) mm, rotated rx -174.06 ry -29.54 rz -11.91 deg; joints [9.131, -47.664, 108.986, -76.339, 63.016, 152.38]
  MoveL 561 to (-201.08, 183.37, -20.25) mm, rotated rx -174.06 ry -29.54 rz -11.91 deg; joints [9.152, -47.8, 109.266, -76.394, 62.991, 152.54]
  MoveL 562 to (-206.05, 183.37, -11.57) mm, rotated rx -174.06 ry -29.54 rz -11.91 deg; joints [8.954, -48.29, 109.337, -76.348, 62.998, 152.058]
  MoveL 563 to (-199.6, 183.37, -8.41) mm, rotated rx -174.06 ry -29.54 rz -11.91 deg; joints [9.207, -48.412, 109.243, -76.036, 63.168, 151.856]
  MoveL 564 to (-197.85, 183.37, -8.4) mm, rotated rx -174.06 ry -29.54 rz -11.91 deg; joints [9.275, -48.4, 109.218, -75.973, 63.204, 151.85]
  MoveL 565 to (-197.85, 183.37, -4.14) mm, rotated rx -174.06 ry -29.54 rz -11.91 deg; joints [9.274, -48.623, 109.215, -75.863, 63.259, 151.605]
  MoveL 566 to (-197.85, 183.24, -3.66) mm, rotated rx -174.06 ry -29.54 rz -11.91 deg; joints [9.275, -48.653, 109.226, -75.853, 63.264, 151.584]
  MoveL 567 to (-197.85, 182.89, -3.31) mm, rotated rx -174.06 ry -29.54 rz -11.91 deg; joints [9.277, -48.686, 109.256, -75.85, 63.265, 151.581]
  MoveL 568 to (-197.85, 182.41, -3.19) mm, rotated rx -174.06 ry -29.54 rz -11.91 deg; joints [9.28, -48.714, 109.298, -75.855, 63.263, 151.597]
  MoveL 569 to (-197.85, 181.14, -3.19) mm, rotated rx -174.06 ry -29.54 rz -11.91 deg; joints [9.289, -48.769, 109.41, -75.876, 63.253, 151.659]
  MoveL 570 to (-197.85, 180.67, -3.31) mm, rotated rx -174.06 ry -29.54 rz -11.91 deg; joints [9.292, -48.783, 109.452, -75.887, 63.248, 151.69]
  MoveL 571 to (-197.85, 180.32, -3.66) mm, rotated rx -174.06 ry -29.54 rz -11.91 deg; joints [9.294, -48.78, 109.483, -75.901, 63.241, 151.728]
  MoveL 572 to (-197.85, 180.19, -4.14) mm, rotated rx -174.06 ry -29.54 rz -11.91 deg; joints [9.295, -48.761, 109.495, -75.916, 63.234, 151.761]
  MoveL 573 to (-197.85, 180.19, -8.4) mm, rotated rx -174.06 ry -29.54 rz -11.91 deg; joints [9.296, -48.538, 109.498, -76.026, 63.179, 152.007]
  MoveL 574 to (-199.6, 180.19, -8.41) mm, rotated rx -174.06 ry -29.54 rz -11.91 deg; joints [9.227, -48.55, 109.523, -76.089, 63.144, 152.013]
  MoveL 575 to (-206.05, 180.19, -11.57) mm, rotated rx -174.06 ry -29.54 rz -11.91 deg; joints [8.974, -48.427, 109.617, -76.402, 62.973, 152.216]
  MoveL 576 to (-201.08, 180.19, -20.25) mm, rotated rx -174.06 ry -29.54 rz -11.91 deg; joints [9.172, -47.936, 109.546, -76.448, 62.967, 152.7]
  MoveL 577 to (-201.08, 177.02, -20.25) mm, rotated rx -174.06 ry -29.54 rz -11.91 deg; joints [9.192, -48.072, 109.825, -76.503, 62.943, 152.859]
  MoveL 578 to (-206.05, 177.02, -11.57) mm, rotated rx -174.06 ry -29.54 rz -11.91 deg; joints [8.994, -48.564, 109.896, -76.457, 62.949, 152.374]
  MoveL 579 to (-199.6, 177.02, -8.41) mm, rotated rx -174.06 ry -29.54 rz -11.91 deg; joints [9.248, -48.687, 109.803, -76.142, 63.119, 152.17]
  MoveL 580 to (-197.85, 177.02, -8.4) mm, rotated rx -174.06 ry -29.54 rz -11.91 deg; joints [9.317, -48.676, 109.777, -76.079, 63.155, 152.164]
  MoveL 581 to (-197.85, 177.02, -4.14) mm, rotated rx -174.06 ry -29.54 rz -11.91 deg; joints [9.316, -48.899, 109.774, -75.968, 63.209, 151.917]
  MoveL 582 to (-197.85, 176.89, -3.66) mm, rotated rx -174.06 ry -29.54 rz -11.91 deg; joints [9.316, -48.93, 109.785, -75.958, 63.214, 151.896]
  MoveL 583 to (-197.85, 176.54, -3.31) mm, rotated rx -174.06 ry -29.54 rz -11.91 deg; joints [9.319, -48.963, 109.815, -75.955, 63.216, 151.893]
  MoveL 584 to (-197.85, 176.06, -3.19) mm, rotated rx -174.06 ry -29.54 rz -11.91 deg; joints [9.322, -48.99, 109.857, -75.959, 63.214, 151.909]
  MoveL 585 to (-197.85, 174.79, -3.19) mm, rotated rx -174.06 ry -29.54 rz -11.91 deg; joints [9.33, -49.046, 109.968, -75.98, 63.204, 151.971]
  MoveL 586 to (-197.85, 174.32, -3.31) mm, rotated rx -174.06 ry -29.54 rz -11.91 deg; joints [9.333, -49.06, 110.01, -75.991, 63.199, 152.002]
  MoveL 587 to (-197.85, 173.97, -3.66) mm, rotated rx -174.06 ry -29.54 rz -11.91 deg; joints [9.335, -49.057, 110.041, -76.006, 63.192, 152.039]
  MoveL 588 to (-197.85, 173.84, -4.14) mm, rotated rx -174.06 ry -29.54 rz -11.91 deg; joints [9.336, -49.037, 110.053, -76.02, 63.185, 152.073]
  MoveL 589 to (-197.85, 173.84, -8.4) mm, rotated rx -174.06 ry -29.54 rz -11.91 deg; joints [9.338, -48.813, 110.056, -76.131, 63.131, 152.321]
  MoveL 590 to (-199.6, 173.84, -8.41) mm, rotated rx -174.06 ry -29.54 rz -11.91 deg; joints [9.268, -48.824, 110.081, -76.195, 63.095, 152.327]
  MoveL 591 to (-206.05, 173.84, -11.57) mm, rotated rx -174.06 ry -29.54 rz -11.91 deg; joints [9.014, -48.701, 110.175, -76.511, 62.925, 152.532]
  MoveL 592 to (-201.08, 173.84, -20.25) mm, rotated rx -174.06 ry -29.54 rz -11.91 deg; joints [9.213, -48.207, 110.104, -76.557, 62.919, 153.018]
  MoveL 593 to (-201.08, 170.67, -20.25) mm, rotated rx -174.06 ry -29.54 rz -11.91 deg; joints [9.233, -48.342, 110.382, -76.611, 62.895, 153.177]
  MoveL 594 to (-206.05, 170.67, -11.57) mm, rotated rx -174.06 ry -29.54 rz -11.91 deg; joints [9.034, -48.837, 110.453, -76.565, 62.902, 152.689]
  MoveL 595 to (-199.6, 170.67, -8.41) mm, rotated rx -174.06 ry -29.54 rz -11.91 deg; joints [9.289, -48.961, 110.359, -76.247, 63.071, 152.484]
  MoveL 596 to (-197.85, 170.67, -8.4) mm, rotated rx -174.06 ry -29.54 rz -11.91 deg; joints [9.358, -48.95, 110.334, -76.184, 63.107, 152.477]
  MoveL 597 to (-197.85, 170.67, -4.14) mm, rotated rx -174.06 ry -29.54 rz -11.91 deg; joints [9.357, -49.175, 110.331, -76.072, 63.161, 152.229]
  Set speed (38.1 mm/s)
  MoveL 598 to (-197.89, 170.67, -3.98) mm, rotated rx -174.06 ry -29.54 rz -11.91 deg; joints [9.356, -49.183, 110.331, -76.07, 63.162, 152.22]
  MoveL 599 to (-198.05, 170.35, -3.7) mm, rotated rx -174.06 ry -29.54 rz -11.91 deg; joints [9.351, -49.213, 110.361, -76.073, 63.16, 152.22]
  Set speed (76.2 mm/s)
  MoveL 600 to (-198.05, 167.81, -3.7) mm, rotated rx -174.06 ry -29.54 rz -11.91 deg; joints [9.368, -49.322, 110.583, -76.115, 63.141, 152.344]
  Set speed (38.1 mm/s)
  MoveL 601 to (-197.89, 167.49, -3.98) mm, rotated rx -174.06 ry -29.54 rz -11.91 deg; joints [9.377, -49.321, 110.609, -76.121, 63.138, 152.375]
  MoveL 602 to (-197.85, 167.49, -4.14) mm, rotated rx -174.06 ry -29.54 rz -11.91 deg; joints [9.378, -49.312, 110.608, -76.124, 63.137, 152.384]
  Set speed (76.2 mm/s)
  MoveL 603 to (-197.85, 167.49, -8.4) mm, rotated rx -174.06 ry -29.54 rz -11.91 deg; joints [9.379, -49.086, 110.611, -76.236, 63.083, 152.634]
  MoveL 604 to (-199.6, 167.49, -8.41) mm, rotated rx -174.06 ry -29.54 rz -11.91 deg; joints [9.31, -49.098, 110.637, -76.3, 63.047, 152.64]
  MoveL 605 to (-206.05, 167.49, -11.57) mm, rotated rx -174.06 ry -29.54 rz -11.91 deg; joints [9.054, -48.973, 110.73, -76.618, 62.878, 152.846]
  MoveL 606 to (-201.08, 167.49, -20.25) mm, rotated rx -174.06 ry -29.54 rz -11.91 deg; joints [9.254, -48.477, 110.66, -76.665, 62.871, 153.335]
  MoveL 607 to (-201.08, 164.32, -20.25) mm, rotated rx -174.06 ry -29.54 rz -11.91 deg; joints [9.275, -48.611, 110.937, -76.719, 62.848, 153.494]
  MoveL 608 to (-206.05, 164.32, -11.57) mm, rotated rx -174.06 ry -29.54 rz -11.91 deg; joints [9.075, -49.109, 111.007, -76.672, 62.855, 153.003]
  MoveL 609 to (-199.6, 164.32, -8.41) mm, rotated rx -174.06 ry -29.54 rz -11.91 deg; joints [9.331, -49.234, 110.914, -76.352, 63.024, 152.796]
  MoveL 610 to (-197.85, 164.32, -8.4) mm, rotated rx -174.06 ry -29.54 rz -11.91 deg; joints [9.4, -49.222, 110.888, -76.288, 63.059, 152.79]
  MoveL 611 to (-197.85, 164.32, -4.14) mm, rotated rx -174.06 ry -29.54 rz -11.91 deg; joints [9.399, -49.449, 110.885, -76.176, 63.113, 152.539]
  Set speed (38.1 mm/s)
  MoveL 612 to (-197.89, 164.32, -3.98) mm, rotated rx -174.06 ry -29.54 rz -11.91 deg; joints [9.398, -49.457, 110.886, -76.173, 63.114, 152.53]
  MoveL 613 to (-198.05, 164, -3.7) mm, rotated rx -174.06 ry -29.54 rz -11.91 deg; joints [9.393, -49.487, 110.915, -76.177, 63.112, 152.53]
  Set speed (76.2 mm/s)
  MoveL 614 to (-198.05, 161.46, -3.7) mm, rotated rx -174.06 ry -29.54 rz -11.91 deg; joints [9.41, -49.596, 111.136, -76.218, 63.094, 152.654]
  Set speed (38.1 mm/s)
  MoveL 615 to (-197.89, 161.14, -3.98) mm, rotated rx -174.06 ry -29.54 rz -11.91 deg; joints [9.419, -49.594, 111.162, -76.225, 63.091, 152.685]
  MoveL 616 to (-197.85, 161.14, -4.14) mm, rotated rx -174.06 ry -29.54 rz -11.91 deg; joints [9.42, -49.585, 111.162, -76.227, 63.09, 152.694]
  Set speed (76.2 mm/s)
  MoveL 617 to (-197.85, 161.14, -8.4) mm, rotated rx -174.06 ry -29.54 rz -11.91 deg; joints [9.422, -49.358, 111.165, -76.34, 63.036, 152.945]
  MoveL 618 to (-199.6, 161.14, -8.41) mm, rotated rx -174.06 ry -29.54 rz -11.91 deg; joints [9.352, -49.37, 111.19, -76.404, 63, 152.952]
  MoveL 619 to (-206.05, 161.14, -11.57) mm, rotated rx -174.06 ry -29.54 rz -11.91 deg; joints [9.095, -49.244, 111.284, -76.725, 62.832, 153.16]
  MoveL 620 to (-201.08, 161.14, -20.25) mm, rotated rx -174.06 ry -29.54 rz -11.91 deg; joints [9.296, -48.746, 111.213, -76.773, 62.825, 153.652]
  MoveL 621 to (-201.08, 157.97, -20.25) mm, rotated rx -174.06 ry -29.54 rz -11.91 deg; joints [9.317, -48.879, 111.489, -76.826, 62.802, 153.81]
  MoveL 622 to (-206.05, 157.97, -11.57) mm, rotated rx -174.06 ry -29.54 rz -11.91 deg; joints [9.116, -49.38, 111.56, -76.779, 62.809, 153.316]
  MoveL 623 to (-199.6, 157.97, -8.41) mm, rotated rx -174.06 ry -29.54 rz -11.91 deg; joints [9.373, -49.506, 111.466, -76.456, 62.977, 153.107]
  MoveL 624 to (-197.85, 157.97, -8.4) mm, rotated rx -174.06 ry -29.54 rz -11.91 deg; joints [9.443, -49.494, 111.441, -76.392, 63.012, 153.101]
  MoveL 625 to (-197.85, 157.97, -4.14) mm, rotated rx -174.06 ry -29.54 rz -11.91 deg; joints [9.442, -49.722, 111.437, -76.278, 63.066, 152.849]
  Set speed (38.1 mm/s)
  MoveL 626 to (-197.89, 157.97, -3.98) mm, rotated rx -174.06 ry -29.54 rz -11.91 deg; joints [9.44, -49.731, 111.438, -76.276, 63.068, 152.839]
  MoveL 627 to (-198.05, 157.65, -3.7) mm, rotated rx -174.06 ry -29.54 rz -11.91 deg; joints [9.436, -49.76, 111.467, -76.279, 63.066, 152.839]
  Set speed (76.2 mm/s)
  MoveL 628 to (-198.05, 155.11, -3.7) mm, rotated rx -174.06 ry -29.54 rz -11.91 deg; joints [9.453, -49.869, 111.688, -76.32, 63.047, 152.963]
  Set speed (38.1 mm/s)
  MoveL 629 to (-197.89, 154.79, -3.98) mm, rotated rx -174.06 ry -29.54 rz -11.91 deg; joints [9.461, -49.867, 111.713, -76.327, 63.044, 152.994]
  MoveL 630 to (-197.85, 154.79, -4.14) mm, rotated rx -174.06 ry -29.54 rz -11.91 deg; joints [9.463, -49.858, 111.713, -76.33, 63.043, 153.003]
  Set speed (76.2 mm/s)
  MoveL 631 to (-197.85, 154.79, -8.4) mm, rotated rx -174.06 ry -29.54 rz -11.91 deg; joints [9.464, -49.63, 111.716, -76.443, 62.989, 153.256]
  MoveL 632 to (-199.6, 154.79, -8.41) mm, rotated rx -174.06 ry -29.54 rz -11.91 deg; joints [9.394, -49.641, 111.741, -76.508, 62.954, 153.262]
  MoveL 633 to (-206.05, 154.79, -11.57) mm, rotated rx -174.06 ry -29.54 rz -11.91 deg; joints [9.136, -49.515, 111.835, -76.832, 62.786, 153.472]
  MoveL 634 to (-201.08, 154.79, -20.25) mm, rotated rx -174.06 ry -29.54 rz -11.91 deg; joints [9.338, -49.013, 111.764, -76.88, 62.779, 153.967]
  MoveL 635 to (-201.08, 151.62, -20.25) mm, rotated rx -174.06 ry -29.54 rz -11.91 deg; joints [9.359, -49.146, 112.039, -76.933, 62.756, 154.125]
  MoveL 636 to (-206.05, 151.62, -11.57) mm, rotated rx -174.06 ry -29.54 rz -11.91 deg; joints [9.157, -49.649, 112.11, -76.885, 62.764, 153.628]
